# B&R Automation Studio project RobotNewEra (part 10)

### HmiKeyControlGlobal.typ - Program interface
```iecst
(********************************************************************
 * COPYRIGHT -- Bernecker + Rainer
 ********************************************************************
 * Program: HmiKeyControl
 * File: HmiKeyControl.typ
 * Author: B&R, International Applications
 * Created: March 16, 2009
 ********************************************************************
 * Data types of program HmiKeyControl
 ********************************************************************)

TYPE
	HmiKeyControlSpace_typ : 	STRUCT
		Enable : BOOL;
		X1 : REAL;
		Y1 : REAL;
		Z1 : REAL;
		X2 : REAL;
		Y2 : REAL;
		Z2 : REAL;
	END_STRUCT;
	HmiKeyControlInputCommand_Type : 	STRUCT
		StartKey : BOOL; (* Start button has been pressed *)
		StopKey : BOOL; (* Stop button has been pressed *)
		EmergencyStopKey : BOOL;
		PageKey : ARRAY[0..MAX_PAGE_KEY_MINUS_ONE]OF BOOL;
		VirFunctionKeyLeft : ARRAY[0..MAX_FUNCTION_KEY_MINUS_ONE]OF BOOL;
		VirFunctionKey : ARRAY[0..MAX_FUNCTION_KEY_MINUS_ONE]OF BOOL;
		FunctionKey : ARRAY[0..MAX_FUNCTION_KEY_MINUS_ONE]OF BOOL;
		PlusKey : ARRAY[0..MAX_PLUS_MINUS_KEY_MINUS_ONE]OF BOOL;
		MinusKey : ARRAY[0..MAX_PLUS_MINUS_KEY_MINUS_ONE]OF BOOL;
		KeySwitch : ARRAY[0..1]OF BOOL;
		Key2nd : BOOL;
		ProgramActive : BOOL;
		Acknowledge : BOOL;
		Reset : BOOL;
		JogMode : BOOL;
		JogEnable : BOOL;
		FeedrateChange : BOOL;
		StepOn : BOOL;
		SaftyKeyRight : BOOL;
		SaftyKeyLeft : BOOL;
		SetPC : BOOL;
		FileSelect : BOOL;
		PosSwitch : BOOL;
	END_STRUCT;
	HmiKeyControlInputPara_Type : 	STRUCT
		JogMode : USINT;
		SystemAddress : UDINT;
		CncAddress : UDINT;
		AxesAddress : UDINT;
		JogAddress : UDINT;
		RecipeAddress : UDINT;
		ErrorAddress : UDINT;
		JoystickXValue : DINT;
		JoystickYValue : DINT;
		JoystickZValue : DINT;
	END_STRUCT;
	HmiKeyControlInput_Type : 	STRUCT
		Parameter : HmiKeyControlInputPara_Type;
		Command : HmiKeyControlInputCommand_Type;
	END_STRUCT;
	HmiKeyControlOutputMon_Type : 	STRUCT
		JogJointVelocity : REAL;
		ToolIndex : USINT;
		JogToolIndex : USINT;
		FileName : STRING[32];
		ModuleType : UDINT;
		PosSelect : UINT;
		ShowPos : ARRAY[0..5]OF REAL;
		JogMode : USINT;
	END_STRUCT;
	HmiKeyControlOutput_Type : 	STRUCT
		Monitor : HmiKeyControlOutputMon_Type;
		Status : HmiKeyControlOutputStatus_Type;
	END_STRUCT;
	HmiKeyControlOutputStatus_Type : 	STRUCT
		Enable : USINT;
		Run : BOOL;
		Error : BOOL;
		Moving : BOOL;
		JogEnable : BOOL;
		RealContinue : BOOL;
		MoveStatus : USINT;
		AutoStatus : USINT;
		StatusIconIndex : USINT;
		SwitchMode : USINT;
		SWLimitsIgnored : ARRAY[0..5]OF BOOL;
		MoveAxis : ARRAY[0..5]OF SINT;
	END_STRUCT;
	HmiKeyControlComponentsType : 	STRUCT
		LayerButtons : HmiKeyCtrlLayerButtonsType;
		LayerLogin : HmiKeyCtrlLayerLoginType;
	END_STRUCT;
	HmiKeyCtrlLayerLoginType : 	STRUCT
		Layer : HmiLayerType;
	END_STRUCT;
	HmiKeyCtrlLayerButtonsType : 	STRUCT
		Layer : HmiLayerType;
		Tabs : HmiTabsType;
		ButtonVMinus : HmiButtonType;
		ButtonVPlus : HmiButtonType;
		ButtonSwitchOn : HmiButtonType;
		ButtonLogin : HmiButtonType;
		ButtonJogBase : HmiButtonType;
		ButtonJogTool : HmiButtonType;
		ButtonJogJoint : HmiButtonType;
		ButtonJogDirect : HmiButtonType;
		ButtonSingle : HmiButtonType;
		ButtonCont : HmiButtonType;
		SliderV : HmiSliderType;
		NumericV : HmiNumericType;
	END_STRUCT;
	HmiKeyControl_Type : 	STRUCT
		Input : HmiKeyControlInput_Type;
		Output : HmiKeyControlOutput_Type;
		Components : HmiKeyControlComponentsType;
	END_STRUCT;
END_TYPE
```

### HmiKeyControlGlobal.var
```iecst
(********************************************************************
 * COPYRIGHT -- Bernecker + Rainer
 ********************************************************************
 * Program: HmiKeyControl
 * File: HmiKeyControl.var
 * Author: B&R, International Applications
 * Created: March 16, 2009
 ********************************************************************
 * Variables of program HmiKeyControl
 ********************************************************************)
VAR CONSTANT
	AXIS_STATUS_BACKWARD : USINT := 2;
	AXIS_STATUS_FORWARD : USINT := 1;
	AXIS_STATUS_NOACTIVE : USINT := 0;
	AXIS_STATUS_WARNING : USINT := 3;
	HANDWHEEL_STATUS_ACTIVE : USINT := 1;
	HANDWHEEL_STATUS_HALT : USINT := 2;
	HANDWHEEL_STATUS_NOACTIVE : USINT := 0;
	HMIKEYCONTROL_CHANGEMODEAUTO : UINT := 150;
	HMIKEYCONTROL_CHANGEMODEDRYRUN : UINT := 190;
	HMIKEYCONTROL_CHANGEMODEHOME : UINT := 200;
	HMIKEYCONTROL_CHANGEMODEJOG : UINT := 170;
	HMIKEYCONTROL_CHANGEMODEMDI : UINT := 160;
	HMIKEYCONTROL_CHANGEMODESIMUL : UINT := 210;
	HMIKEYCONTROL_CHANGEMODESINGLE : UINT := 180;
	HMIKEYCONTROL_IDLE : UINT := 100;
	HMIKEYCONTROL_INIT : UINT := 0;
	HMIKEYCONTROL_SELECTAXIS : UINT := 120;
	HMIKEYCONTROL_SELECTFUNCTIONM : UINT := 130;
	HMIKEYCONTROL_SELECTSCALE : UINT := 140;
	HMIKEYCONTROL_SELECTSYSTEM : UINT := 110;
	HMIKEYCONTROL_START : UINT := 220;
	HMIKEYCONTROL_STOPAUTO : UINT := 230;
	HMIKEYCONTROL_STOPDRYRUN : UINT := 231;
	HMIKEYCONTROL_STOPHOME : UINT := 232;
	HMIKEYCONTROL_STOPJOG : UINT := 233;
	HMIKEYCONTROL_STOPMDI : UINT := 234;
	HMIKEYCONTROL_STOPSIMUL : UINT := 235;
	HMIKEYCONTROL_STOPSINGLE : UINT := 236;
	MFUNCTION_M10 : USINT := 10;
	MFUNCTION_M11 : USINT := 11;
	MFUNCTION_M12 : USINT := 12;
	MFUNCTION_M13 : USINT := 13;
	MFUNCTION_M14 : USINT := 14;
	MFUNCTION_M15 : USINT := 15;
	MFUNCTION_M16 : USINT := 16;
	MFUNCTION_M17 : USINT := 17;
	MFUNCTION_COOLING : USINT := 1;
	MFUNCTION_DISABLE : USINT := 2;
	MFUNCTION_RUNNING : USINT := 3;
	MFUNCTION_SPINDLE : USINT := 3;
	MFUNCTION_STANDBY : USINT := 0;
	MFUNCTION_STANDBYRUNNING : USINT := 1;
	MFUNCTION_TIMEPRESSED : TIME := T#2s;
	MFUNCTION_WARNING : USINT := 4;
	MODE_AUTOMATIC : USINT := 0;
	MODE_DRYRUN : USINT := 4;
	MODE_HOME : USINT := 5;
	MODE_MDI : USINT := 1;
	MODE_MOTION_AUTO : USINT := 1;
	MODE_MOTION_JOG : USINT := 0;
	MODE_NOMODE : USINT := 254;
	MODE_SIMULATION : USINT := 6;
	MODE_SINGLESTEP : USINT := 3;
	SCALE_STATUS_ACIVE : BOOL := TRUE;
	SCALE_STATUS_NOACTIVE : BOOL := FALSE;
	SCALE_UNITS_INDEX_0 : REAL := 1.0;
	SCALE_UNITS_INDEX_1 : REAL := 0.1;
	SCALE_UNITS_INDEX_2 : REAL := 0.01;
	SYSTEM_STATUS_NOACTIVE : USINT := 0;
	SYSTEM_STATUS_PROGRAMHALT : USINT := 4;
	SYSTEM_STATUS_RUNNING : USINT := 2;
	SYSTEM_STATUS_SELECTED : USINT := 1;
	SYSTEM_STATUS_SELECTRUNNING : USINT := 3;
	SYSTEM_STATUS_WARNING : USINT := 5;
	JOG_MODE_JOINT : USINT := 0;
	JOG_MODE_BASE : USINT := 1;
	JOG_MODE_TOOL : USINT := 2;
	JOG_MODE_DIRECT : USINT := 3;
	WARNING_TIMEACTIVE : TIME := T#3s;
END_VAR
VAR
	HmiKeyControl : HmiKeyControl_Type := (0);
END_VAR
```

### Program Logical/HmiHandling/HmiKeyCtrl/HmiKeyCtrl (IEC) - Handles the Cnc panel key control  functionalities

#### HmiKeyControlActions.st
```iecst
(*Copy all inputs for this program*)
ACTION HmiKeyControlInputs: //Control all the Inputs

	(* Checks if the Simulation key is active and assignes the commands *)
	IF (HmiKeyControl.Output.Monitor.ModuleType = ARSIM_PC)THEN

		FOR i := 0 TO MAX_FUNCTION_KEY_MINUS_ONE DO
			HmiKeyControl.Input.Command.FunctionKey[i]	:= HmiHardKey.Input.MP50_SimKey[22+i];
		END_FOR

		FOR i := 0 TO MAX_PLUS_MINUS_KEY_MINUS_ONE DO
			HmiKeyControl.Input.Command.PlusKey[i]	:= HmiHardKey.Input.MP50_SimKey[16+i];
		END_FOR

		FOR i := 0 TO MAX_PLUS_MINUS_KEY_MINUS_ONE DO
			HmiKeyControl.Input.Command.MinusKey[i]	:= HmiHardKey.Input.MP50_SimKey[8+i];
		END_FOR

		FOR i := 0 TO MAX_PAGE_KEY_MINUS_ONE DO
			HmiKeyControl.Input.Command.PageKey[i]	:= HmiHardKey.Input.MP50_SimKey[i];
		END_FOR
		HmiKeyControl.Input.Command.PageKey[3] := HmiHardKey.Input.MP50_SimKey[3] OR HmiKeyControl.Input.Command.FileSelect;

		HmiKeyControl.Input.Command.StartKey			:= HmiHardKey.Input.MP50_SimKey[7];
		HmiKeyControl.Input.Command.StopKey 			:= HmiHardKey.Input.MP50_SimKey[15];
		HmiKeyControl.Input.Command.EmergencyStopKey 	:= DI1.I3;
		HmiKeyControl.Input.Command.Key2nd 				:= HmiHardKey.Input.MP50_SimKey[14];
		HmiKeyControl.Input.Command.KeySwitch[JOG] 		:= HmiHardKey.Input.MP50_SimKey[35];
		HmiKeyControl.Input.Command.KeySwitch[AUTO] 	:= HmiHardKey.Input.MP50_SimKey[36];

		HmiKeyControl.Input.Command.SaftyKeyLeft	;
		HmiKeyControl.Input.Command.SaftyKeyRight	;

		HmiKeyControl.Input.Command.SaftyKeyLeft		:= TRUE;
		HmiKeyControl.Input.Command.SaftyKeyRight		:= TRUE;

		HmiHardKey.Input.Joystick_XValue	:= 500;
		HmiHardKey.Input.Joystick_YValue	:= 500;
		HmiHardKey.Input.Joystick_ZValue	:= 500;
	ELSE
		FOR i := 0 TO MAX_FUNCTION_KEY_MINUS_ONE DO
			HmiKeyControl.Input.Command.FunctionKey[i]	:= HmiHardKey.Input.MP50_Key[22+i];
		END_FOR

		FOR i := 0 TO MAX_PLUS_MINUS_KEY_MINUS_ONE DO
			HmiKeyControl.Input.Command.PlusKey[i]	:= HmiHardKey.Input.MP50_Key[16+i];
		END_FOR

		FOR i := 0 TO MAX_PLUS_MINUS_KEY_MINUS_ONE DO
			HmiKeyControl.Input.Command.MinusKey[i]	:= HmiHardKey.Input.MP50_Key[8+i];
		END_FOR

		FOR i := 0 TO MAX_PAGE_KEY_MINUS_ONE DO
			HmiKeyControl.Input.Command.PageKey[i]	:= HmiHardKey.Input.MP50_Key[i];
		END_FOR
		HmiKeyControl.Input.Command.PageKey[3] := HmiHardKey.Input.MP50_Key[3] OR HmiKeyControl.Input.Command.FileSelect;

		HmiKeyControl.Input.Command.StartKey			:= HmiHardKey.Input.MP50_Key[7];
		HmiKeyControl.Input.Command.StopKey 			:= HmiHardKey.Input.MP50_Key[15];
		HmiKeyControl.Input.Command.EmergencyStopKey 	:= DI1.I3;
		HmiKeyControl.Input.Command.Key2nd 				:= HmiHardKey.Input.MP50_Key[14];
		HmiKeyControl.Input.Command.KeySwitch[JOG] 		:= HmiHardKey.Input.MP50_Key[35];
		HmiKeyControl.Input.Command.KeySwitch[AUTO] 	:= HmiHardKey.Input.MP50_Key[36];

		HmiKeyControl.Input.Command.SaftyKeyLeft		:= DI1.I1;
		HmiKeyControl.Input.Command.SaftyKeyRight		:= DI1.I2;

		HmiKeyControl.Input.Command.SaftyKeyLeft		:= TRUE;
		HmiKeyControl.Input.Command.SaftyKeyRight		:= TRUE;
	END_IF

	HmiKeyControl.Input.Parameter.JoystickXValue	:= HmiHardKey.Input.Joystick_XValue;
	HmiKeyControl.Input.Parameter.JoystickYValue	:= HmiHardKey.Input.Joystick_YValue;
	HmiKeyControl.Input.Parameter.JoystickZValue	:= HmiHardKey.Input.Joystick_ZValue;

	//LEDs
	HmiHardKey.Output.Motion_Led 		:= pSystem[0].Output.Status.ControllerStatus <> 0;
	HmiHardKey.Output.Run_Led 			:= 1;
	HmiHardKey.Output.Error_Led 		:= HmiKeyControl.Output.Status.Error;
	HmiHardKey.Output.Process_Led 		:= pCnc[0].Output.State.Moving;

END_ACTION

ACTION HmiKeyControlStateHandling: // Main State Machine

	// Emegency Stop
	IF pSystem[0].Output.State.Errorstop THEN
		Internal.HmiKeyControlState := HMIKEYCONSTATESTEP_ERROR;
	END_IF

	// Switch On/Off Control
	IF HmiKeyControl.Components.LayerButtons.ButtonSwitchOn.Value > HmiKeyControl.Components.LayerButtons.ButtonSwitchOn.OldValue THEN
		IF 	pSystem[0].Output.State.Disabled THEN
			pSystem[0].Input.Command.Enable := 1;
			Internal.HmiKeyControlState := HMIKEYCONSTATESTEP_DISABLED;
		ELSIF pCnc[0].Output.State.Standby THEN
			pSystem[0].Input.Command.Enable := 0;
		END_IF
	END_IF

	CASE Internal.HmiKeyControlState OF

		HMIKEYCONSTATESTEP_DISABLED:

			IF HmiKeyControl.Components.LayerButtons.ButtonSwitchOn.Value > HmiKeyControl.Components.LayerButtons.ButtonSwitchOn.OldValue AND NOT pSystem[0].Output.Status.Busy THEN

				IF 	pSystem[0].Output.State.Disabled THEN
					pSystem[0].Input.Command.Enable := 1;
					Internal.HmiKeyControlState := HMIKEYCONSTATESTEP_HOME;
				ELSIF pCnc[0].Output.State.Standby THEN
					pSystem[0].Input.Command.Enable := 0;
				END_IF

			END_IF

			// If Press Start when disabled, show the warning
			IF (HmiKeyControl.Input.Command.StartKey > Internal.OldCommand.StartKey) THEN

				WarnMessage[0] := 1;

			END_IF

		HMIKEYCONSTATESTEP_HOME: (* Homing Axes *)

			// Do the homing, homing position is stored in the Recipe
			IF NOT pSystem[0].Output.Status.Busy AND pSystem[0].Output.Status.ControllerStatus <> 0 THEN

				FOR i := 6 TO MAX_AX_MINUS_TWO DO
					pAxes[i].Input.Parameter.HomePosition := pRecipe.Data.System.HomePosition[i];
				END_FOR

				pSystem[0].Input.Command.Home := 1;

				Internal.HmiKeyControlState := HMIKEYCONSTATESTEP_CHANGEMODE;

			END_IF

		HMIKEYCONSTATESTEP_CHANGEMODE: (* Actual Standby State(After Homing) *)

			IF NOT pSystem[0].Output.Status.Busy AND pSystem[0].Input.Command.Home = 0 THEN

				// Just to avoid the sw limits being ignored
				FOR i := 6 TO MAX_AX_MINUS_TWO DO

					IF HmiKeyControl.Output.Status.SWLimitsIgnored[i - 6] THEN
						pAxes[i].Input.Parameter.WriteParID := ACP10PAR_SGEN_SW_END_IGNORE;
						pAxes[i].Input.Parameter.WriteParIDText := '0';
						pAxes[i].Input.Command.WriteAxisPar := 1;
					END_IF

					HmiKeyControl.Output.Status.SWLimitsIgnored[i - 6] := FALSE;

				END_FOR

				// Make Sure the robot is homed before mode switch to CNC
				IF HmiRetain.HmiKeyControl.MechHomeOK THEN

					IF HmiKeyControl.Output.Status.SwitchMode = LOCK THEN

						pSystem[0].Input.Parameter.Mode := 1;
						Internal.HmiKeyControlState := HMIKEYCONSTATESTEP_ACTIVE_JOG; // JOG MEANS NO CNC, not the Jog Mode for Robot (This mode is for Setting home position)

					ELSE

						pSystem[0].Input.Parameter.Mode := 0;
						Internal.HmiKeyControlState := HMIKEYCONSTATESTEP_ACTIVE_AUTO; // AUTO MEANS CNC, including Jog Mode and Auto Mode

					END_IF

				ELSE

					pSystem[0].Input.Parameter.Mode := 1;
					Internal.HmiKeyControlState := HMIKEYCONSTATESTEP_ACTIVE_JOG;

				END_IF

				pSystem[0].Input.Command.ChangeMode := 1;

			END_IF

		HMIKEYCONSTATESTEP_ACTIVE_JOG:

			IF pSystem[0].Output.Monitor.Mode = 1 THEN (* 1 for No CNC and 0 for CNC *)

				IF HmiKeyControl.Output.Status.SwitchMode <> LOCK THEN

					IF HmiRetain.HmiKeyControl.MechHomeOK THEN

						pSystem[0].Input.Parameter.Mode := 0;
						pSystem[0].Input.Command.ChangeMode := 1;

						StartState := 0;

						Internal.HmiKeyControlState := HMIKEYCONSTATESTEP_ACTIVE_AUTO;

					END_IF

				END_IF

				// The Moving Of Axis in NON-CNC Mode is only allowed in PAGE_SETUPCALIB
				IF HmiGlobal.PageControl.ActPage = PAGE_SETUPCALIB AND pSystem[0].Output.State.Active THEN

					FOR i := 0 TO 5 DO
						(* For MP50-4*)
						IF HmiSetupCtrl.Components.PageCalib.LayerDefault.ButtonAxisToggle[i].Value = 1 THEN // Only when certain Axis is toggled(only one axis will be toggled at one time)
							// Using MCMoveVelocity(Axis Controlling) for Calibration
							IF EDGEPOS((HmiKeyControl.Input.Command.SaftyKeyLeft OR HmiKeyControl.Input.Command.SaftyKeyRight) AND (HmiKeyControl.Input.Command.PlusKey[i] <> 0)
								) THEN
								pAxes[i+6].Input.Parameter.Velocity := HmiKeyControl.Components.LayerButtons.SliderV.Value /100.0 * pRecipe.Data.System.JointJogSpeed;
								pAxes[i+6].Input.Parameter.Direction := mcPOSITIVE_DIR;
								pAxes[i+6].Input.Command.MoveVelocity := 1;
							ELSIF EDGENEG((HmiKeyControl.Input.Command.SaftyKeyLeft OR HmiKeyControl.Input.Command.SaftyKeyRight) AND (HmiKeyControl.Input.Command.PlusKey[i] <> 0)
								) THEN
								pAxes[i+6].Input.Command.Stop := 1;
							ELSIF EDGEPOS((HmiKeyControl.Input.Command.SaftyKeyLeft OR HmiKeyControl.Input.Command.SaftyKeyRight) AND (HmiKeyControl.Input.Command.MinusKey[i] <> 0)
								) THEN
								pAxes[i+6].Input.Parameter.Velocity := HmiKeyControl.Components.LayerButtons.SliderV.Value /100.0 * pRecipe.Data.System.JointJogSpeed;
								pAxes[i+6].Input.Parameter.Direction := mcNEGATIVE_DIR;
								pAxes[i+6].Input.Command.MoveVelocity := 1;
							ELSIF EDGENEG((HmiKeyControl.Input.Command.SaftyKeyLeft OR HmiKeyControl.Input.Command.SaftyKeyRight) AND (HmiKeyControl.Input.Command.MinusKey[i] <> 0)
								) THEN
								pAxes[i+6].Input.Command.Stop := 1;

							END_IF
						ELSE

							// Otherweise stop the Movement
							IF pAxes[i+6].Output.State.ContinuousMotion THEN

								pAxes[i+6].Input.Command.Stop := 1;

							END_IF
						END_IF

					END_FOR

				ELSE
					// In other Page stop the Axis Any Way
					FOR i := 0 TO 5 DO
						IF pAxes[i+6].Output.State.ContinuousMotion THEN

							pAxes[i+6].Input.Command.Stop := 1;

						END_IF
					END_FOR
				END_IF

			END_IF

		HMIKEYCONSTATESTEP_ACTIVE_AUTO:  // CNC Mode

			IF pSystem[0].Output.Monitor.Mode = 0 THEN
				// Change to Non-CNC Mode
				IF HmiKeyControl.Output.Status.SwitchMode = LOCK THEN

					pSystem[0].Input.Parameter.Mode := 1;
					pSystem[0].Input.Command.ChangeMode := 1;

					Internal.HmiKeyControlState := HMIKEYCONSTATESTEP_ACTIVE_JOG;

				END_IF

				(* UserLevel higher than 0 and Mode is Auto then Start OR Stop is allowed *)
				IF pSystem[0].Output.State.Active AND gUserLevel > 0 AND HmiKeyControl.Output.Status.MoveStatus = AUTO THEN

					pCnc[0].Input.Parameter.NcInitProgramName := '';

					(* Stop the Program: Once for Halt, Twice for Stop *)
					IF HmiKeyControl.Input.Command.StopKey > Internal.OldCommand.StopKey THEN

						IF pCnc[0].Output.State.Moving AND NOT pCnc[0].Output.Status.Halted THEN
							pCnc[0].Input.Command.Halt := 1;
						ELSE
							pCnc[0].Input.Command.Stop := 1;
						END_IF

					END_IF

					// Start the program
					IF (HmiKeyControl.Input.Command.StartKey > Internal.OldCommand.StartKey) THEN

						(* if halted continue else start *)
						IF pCnc[0].Output.Status.Halted THEN
							pCnc[0].Input.Command.Continue := 1;
						ELSE

							IF HmiRetain.HmiProgram.Name <> ''  THEN
								IF HmiRetain.HmiProgram.Ptr <> 0 THEN // Start the Program from some line (Not working right now)
									brsitoa(HmiRetain.HmiProgram.Ptr, ADR(TempStr));
									pCnc[0].Input.Parameter.NcProgramName := CONCAT(CONCAT(CONCAT(HmiRetain.HmiProgram.Name, '.st'), '::'), TempStr);
								ELSE
									pCnc[0].Input.Parameter.NcProgramName := CONCAT(HmiRetain.HmiProgram.Name, '.st');
								END_IF

								pCnc[0].Input.Parameter.NcProgramStartPos := -1;
								pCnc[0].Input.Parameter.NcProgramStartMode := ncFILE;
								pCnc[0].Input.Command.StartNcProgram := 1;

							END_IF
						END_IF

					END_IF

					//If Program is stopped, reset the Pointer
					IF EDGENEG(pCnc[0].Output.State.Moving) THEN

						HmiRetain.HmiProgram.Ptr := 0;

					END_IF

				END_IF

			ELSIF pSystem[0].Output.State.Standby AND pSystem[0].Output.Status.HomingOk THEN

				Internal.HmiKeyControlState := HMIKEYCONSTATESTEP_CHANGEMODE;

			END_IF

		HMIKEYCONSTATESTEP_ERROR:
			// Press the Stop key in Error state means reset the error
			IF (HmiKeyControl.Input.Command.StopKey > Internal.OldCommand.StopKey) THEN
				pSystem[0].Input.Command.Reset := 1;
			END_IF

			pCncDat ACCESS pCnc[0].Output.Monitor.CncAddress;

			(* In Case Cnc Still Runing even in Errorstop State *)
			IF (pCncDat.move.status.cnt_ncprog <> 0) THEN
				ncaction(ADR(pCncDat), ncMOVE, ncSTOP);
			END_IF

			IF NOT pSystem[0].Output.State.Errorstop THEN
				IF pSystem[0].Output.Status.HomingOk THEN
					Internal.HmiKeyControlState := HMIKEYCONSTATESTEP_CHANGEMODE;
				ELSE
					Internal.HmiKeyControlState := HMIKEYCONSTATESTEP_HOME;
				END_IF

			END_IF

	END_CASE

	// SingleStep Control
	IF pCnc[0].Output.State.Standby THEN
		(* Switch between Modes: *)
		IF (HmiKeyControl.Components.LayerButtons.ButtonSingle.Value > HmiKeyControl.Components.LayerButtons.ButtonSingle.OldValue) THEN
			IF NOT pCnc[0].Output.Status.SingleStep THEN
				pCnc[0].Input.Command.StartSingleStep := 1;
			END_IF
		END_IF

		IF (HmiKeyControl.Components.LayerButtons.ButtonCont.Value > HmiKeyControl.Components.LayerButtons.ButtonCont.OldValue) THEN
			IF pCnc[0].Output.Status.SingleStep THEN
				pCnc[0].Input.Command.StopSingleStep := 1;
			END_IF
		END_IF

		// Switch off Single Step for Jog
		IF HmiKeyControl.Output.Status.MoveStatus = JOG AND pCnc[0].Output.Status.SingleStep THEN
			pCnc[0].Input.Command.StopSingleStep := 1;
		END_IF

	END_IF
	// Show different Pics
	HmiKeyControl.Components.LayerButtons.Tabs.ButtonsTab[0].BmpIdx := pCnc[0].Output.Status.SingleStep;

END_ACTION

ACTION HmiKeyControlJog: // Jog Control

	IF gUserLevel = 0 THEN

		pJog.Run 	:= 0;

	ELSE
		// Four Modes Available: TOOL; BASE; JOINT; DIRECT
		IF pCnc[0].Output.State.Standby THEN
			(* Switch between Modes *)
			IF HmiKeyControl.Components.LayerButtons.ButtonJogTool.Value > HmiKeyControl.Components.LayerButtons.ButtonJogTool.OldValue THEN
				HmiKeyControl.Input.Parameter.JogMode := JOG_MODE_TOOL;
			END_IF

			IF HmiKeyControl.Components.LayerButtons.ButtonJogBase.Value > HmiKeyControl.Components.LayerButtons.ButtonJogBase.OldValue THEN
				HmiKeyControl.Input.Parameter.JogMode := JOG_MODE_BASE;
			END_IF

			IF HmiKeyControl.Components.LayerButtons.ButtonJogJoint.Value > HmiKeyControl.Components.LayerButtons.ButtonJogJoint.OldValue THEN
				HmiKeyControl.Input.Parameter.JogMode := JOG_MODE_JOINT;
			END_IF

			IF HmiKeyControl.Components.LayerButtons.ButtonJogDirect.Value > HmiKeyControl.Components.LayerButtons.ButtonJogDirect.OldValue THEN
				HmiKeyControl.Input.Parameter.JogMode := JOG_MODE_DIRECT;
			END_IF

		END_IF
		// Show Different Pics
		HmiKeyControl.Components.LayerButtons.Tabs.ButtonsTab[2].BmpIdx := HmiKeyControl.Input.Parameter.JogMode;

		// Buttons Control (+/- Buttons) Plus/Minuskey -> MoveAxis
		IF HmiKeyControl.Output.Status.MoveStatus = JOG THEN

			FOR i := 0 TO 5 DO
				(* For MP50-4*)
				IF (HmiKeyControl.Input.Command.PlusKey[i] <> 0)  THEN
					HmiKeyControl.Output.Status.MoveAxis[i] := 1;
				ELSIF (HmiKeyControl.Input.Command.MinusKey[i] <> 0) THEN
					HmiKeyControl.Output.Status.MoveAxis[i] := -1;
				ELSE
					HmiKeyControl.Output.Status.MoveAxis[i] := 0;
				END_IF

			END_FOR

			IF (HmiKeyControl.Input.Command.SaftyKeyLeft = 0)
				AND (HmiKeyControl.Input.Command.SaftyKeyRight = 0) THEN

				HmiKeyControl.Output.Status.MoveAxis[0] := 0;
				HmiKeyControl.Output.Status.MoveAxis[1] := 0;
				HmiKeyControl.Output.Status.MoveAxis[2] := 0;
				HmiKeyControl.Output.Status.MoveAxis[3] := 0;
				HmiKeyControl.Output.Status.MoveAxis[4] := 0;
				HmiKeyControl.Output.Status.MoveAxis[5] := 0;
			END_IF

			IF (HmiKeyControl.Output.Status.MoveAxis[0] <> 0) OR
				(HmiKeyControl.Output.Status.MoveAxis[1] <> 0) OR
				(HmiKeyControl.Output.Status.MoveAxis[2] <> 0) OR
				(HmiKeyControl.Output.Status.MoveAxis[3] <> 0) OR
				(HmiKeyControl.Output.Status.MoveAxis[4] <> 0) OR
				(HmiKeyControl.Output.Status.MoveAxis[5] <> 0) THEN

				IF (pRecipe.Data.System.JointJogSpeed <> 0) THEN

					IF (HmiKeyControl.Input.Parameter.JogMode = JOG_MODE_BASE) THEN
						pJog.Speed 	:= pRecipe.Data.System.PathJogSpeed;

					ELSIF (HmiKeyControl.Input.Parameter.JogMode = JOG_MODE_TOOL) THEN
						pJog.Speed 	:= pRecipe.Data.System.PathJogSpeed;

					ELSIF (HmiKeyControl.Input.Parameter.JogMode = JOG_MODE_JOINT) THEN
						pJog.Speed 	:= pRecipe.Data.System.JointJogSpeed;
					END_IF

					pJog.Mode	:= HmiKeyControl.Input.Parameter.JogMode;
					pJog.Run 	:= 1;

				END_IF

			ELSE

				// Special Control For Direct Mode
				IF (HmiKeyControl.Input.Command.SaftyKeyLeft = 1 OR HmiKeyControl.Input.Command.SaftyKeyRight = 1) AND
					HmiKeyControl.Input.Parameter.JogMode = JOG_MODE_DIRECT AND HmiGlobal.PageControl.ActPage = PAGE_JOGGING AND
					HmiJog.Components.LayerDefault.TextActSet.TextIndex = 1 THEN // The use of this mode is restricted to certain page and certain status

					IF HmiJog.Components.LayerDefault.ButtonCheckVar.Value = 0 THEN // Use the point from numeric inputs.
						IF HmiJog.Components.LayerDefault.DropdownJointTCP.SelectedIndex = 0 THEN

							pJog.Speed := pRecipe.Data.System.JointJogSpeed;

							JointSync.JointAxis[0] := HmiJog.Components.LayerDefault.NumericPosSet[0].Value;
							JointSync.JointAxis[1] := HmiJog.Components.LayerDefault.NumericPosSet[1].Value;
							JointSync.JointAxis[2] := HmiJog.Components.LayerDefault.NumericPosSet[2].Value;
							JointSync.JointAxis[3] := HmiJog.Components.LayerDefault.NumericPosSet[3].Value;
							JointSync.JointAxis[4] := HmiJog.Components.LayerDefault.NumericPosSet[4].Value;
							JointSync.JointAxis[5] := HmiJog.Components.LayerDefault.NumericPosSet[5].Value;

							JointTCPSync := 1;

						ELSE
							pJog.Speed := pRecipe.Data.System.PathJogSpeed;

							PointSync.Pos.x := HmiJog.Components.LayerDefault.NumericPosSet[0].Value;
							PointSync.Pos.y := HmiJog.Components.LayerDefault.NumericPosSet[1].Value;
							PointSync.Pos.z := HmiJog.Components.LayerDefault.NumericPosSet[2].Value;
							PointSync.Orient.Angle[0] := HmiJog.Components.LayerDefault.NumericPosSet[3].Value;
							PointSync.Orient.Angle[1] := HmiJog.Components.LayerDefault.NumericPosSet[4].Value;
							PointSync.Orient.Angle[2] := HmiJog.Components.LayerDefault.NumericPosSet[5].Value;
							PointSync.Orient.Angle[3] := HmiJog.Components.LayerDefault.NumericPosSet[6].Value;

							IF HmiJog.Components.LayerDefault.DropdownEulerQuan.SelectedIndex = 1 THEN
								PointSync.Orient.Type := MX_QUATERNION;
							ELSE
								PointSync.Orient.Type := 1;
							END_IF

							JointTCPSync := 0;
						END_IF
					ELSE
						// Else use the Point from the File
						IF HmiRetain.HmiJog.Device = HmiRetain.HmiEditor.Device AND HmiRetain.HmiJog.Name = HmiRetain.HmiEditor.Name THEN

							IF HmiRetain.HmiJog.Joint.Set THEN

								pJog.Speed := pRecipe.Data.System.JointJogSpeed;

								JointSync := HmiRetain.HmiJog.Joint.Joint;

								JointTCPSync := 1;

							END_IF

							IF HmiRetain.HmiJog.Point.Set THEN

								pJog.Speed := pRecipe.Data.System.PathJogSpeed;

								PointSync := HmiRetain.HmiJog.Point.Point;

								JointTCPSync := 0;

							END_IF

						END_IF

					END_IF

					pJog.Mode	:= HmiKeyControl.Input.Parameter.JogMode;

					pJog.Run 	:= 1;

				ELSE

					pJog.Run	:= 0;

				END_IF

			END_IF

		END_IF

	END_IF

END_ACTION

ACTION HmiKeyControlStatus:

	// Control all the status, altogether 4  stats(Disabled/LOCK/JOG/AUTO)
	IF HmiKeyControl.Input.Command.KeySwitch[JOG] THEN
		HmiKeyControl.Output.Status.SwitchMode := JOG;
	ELSIF HmiKeyControl.Input.Command.KeySwitch[AUTO] THEN
		HmiKeyControl.Output.Status.SwitchMode := AUTO;
	ELSE
		HmiKeyControl.Output.Status.SwitchMode := LOCK;
	END_IF

	IF pSystem[0].Output.State.Disabled THEN // Not Enabled = DISABLED
		HmiKeyControl.Output.Status.MoveStatus := DISABLED;
	ELSE
		IF pSystem[0].Output.Monitor.Mode = 1 THEN // If in the middle, Lock
			HmiKeyControl.Output.Status.MoveStatus := LOCK;
		ELSIF pSystem[0].Output.Monitor.Mode = 0 THEN // Left Jog
			IF HmiKeyControl.Output.Status.SwitchMode = AUTO THEN
				HmiKeyControl.Output.Status.MoveStatus := AUTO;
			ELSE // Right Auto
				HmiKeyControl.Output.Status.MoveStatus := JOG;
			END_IF

		END_IF

	END_IF
	// In AutoMode 3 Status(RUN/PAUSE/STOP)
	IF (HmiKeyControl.Output.Status.MoveStatus = AUTO) THEN
		IF (pCnc[0].Output.State.Moving = 1) AND (pCnc[0].Output.Status.Halted  = 0) THEN
			HmiKeyControl.Output.Status.AutoStatus := RUN;
		ELSIF (pCnc[0].Output.State.Moving = 1) AND (pCnc[0].Output.Status.Halted  = 1) THEN
			HmiKeyControl.Output.Status.AutoStatus := PAUSE;
		ELSE
			HmiKeyControl.Output.Status.AutoStatus := STOP;
		END_IF
	ELSE
		HmiKeyControl.Output.Status.AutoStatus := STOP;
	END_IF

END_ACTION

ACTION HmiKeyControlPage:
	// Turn the Pages
	IF (HmiKeyControl.Input.Command.PageKey[0] > Internal.OldCommand.PageKey[0]) THEN
		HmiGlobal.PageControl.SetPage := PAGE_MAIN;
	END_IF

	IF (HmiKeyControl.Input.Command.PageKey[1] > Internal.OldCommand.PageKey[1]) AND (gUserLevel >= 1) THEN
		HmiGlobal.PageControl.SetPage := PAGE_SETUP;
	END_IF

	IF (HmiKeyControl.Input.Command.PageKey[2] > Internal.OldCommand.PageKey[2]) AND (gUserLevel >= 1) THEN
		HmiGlobal.PageControl.SetPage := PAGE_IO;
	END_IF

	IF (HmiKeyControl.Input.Command.PageKey[3] > Internal.OldCommand.PageKey[3]) AND (gUserLevel >= 1) THEN
		HmiGlobal.PageControl.SetPage := PAGE_PROGRAM;
	END_IF

	// Edit Page cannot be entered if no Program available
	IF (HmiKeyControl.Input.Command.PageKey[4] > Internal.OldCommand.PageKey[4]) AND (gUserLevel >= 1) AND
		HmiRetain.HmiEditor.Device <> '' AND HmiRetain.HmiEditor.Name <> ''  THEN
		HmiGlobal.PageControl.SetPage := PAGE_EDITOR;
	END_IF

	IF (HmiKeyControl.Input.Command.PageKey[5] > Internal.OldCommand.PageKey[5]) AND (gUserLevel >= 1) THEN
		HmiGlobal.PageControl.SetPage := PAGE_JOGGING;
	END_IF

	IF (HmiKeyControl.Input.Command.PageKey[6] > Internal.OldCommand.PageKey[6]) AND (gUserLevel >= 1) THEN
		HmiGlobal.PageControl.SetPage := PAGE_ALARM;
	END_IF

	// If userlevel < 1, robot is disabled
	IF (gUserLevel < 1) THEN

		HmiKeyControl.Components.LayerButtons.ButtonSwitchOn.Value := 0;

	END_IF

	IF HmiKeyControl.Components.LayerButtons.ButtonLogin.Value > HmiKeyControl.Components.LayerButtons.ButtonLogin.OldValue THEN

		HmiKeyControl.Components.LayerLogin.Layer.StatusDatapoint := 0;

	END_IF

END_ACTION

ACTION HmiKeyControlFeedOverride:

	// Using 1st Order Filter to smoothe the Feedrate to avoid rash change.
	LCRPT1_0(enable := 1 , x := HmiKeyControl.Components.LayerButtons.SliderV.Value / 100.0, t := 1); // Time constant 1 second
	pCnc[0].Input.Parameter.FeedrateOverride := LCRPT1_0.y;
	pCnc[0].Input.Parameter.RapidOverride		:= pCnc[0].Input.Parameter.FeedrateOverride;

	// Visual Effect of Slider of Feedrate
	IF NOT pCnc[0].Output.State.Moving OR pCnc[0].Output.Status.Halted THEN
		HmiKeyControl.Components.LayerButtons.SliderV.StatusDatapoint := BIT_SET(HmiKeyControl.Components.LayerButtons.SliderV.StatusDatapoint, 1);
	ELSE
		HmiKeyControl.Components.LayerButtons.SliderV.StatusDatapoint := BIT_CLR(HmiKeyControl.Components.LayerButtons.SliderV.StatusDatapoint, 1);
	END_IF

	(* Delicate control of Plus/Minus Button --- Done by Others(MB Kai YH) *)
	IF (HmiKeyControl.Components.LayerButtons.ButtonVPlus.Value > HmiKeyControl.Components.LayerButtons.ButtonVPlus.OldValue) THEN
		HmiKeyControl.Components.LayerButtons.SliderV.Value := HmiKeyControl.Components.LayerButtons.SliderV.Value + 1;
		VPlus1T := VPlus1T + cycT;
		VPlus10T := VPlus10T + cycT;
	ELSIF (HmiKeyControl.Components.LayerButtons.ButtonVPlus.Value <> 0)
		AND (HmiKeyControl.Components.LayerButtons.ButtonVPlus.OldValue <> 0) THEN
		VPlus1T := VPlus1T + cycT;
		VPlus10T := VPlus10T + cycT;

		IF (VPlus10T > (10*CalculateInterval))
			AND (VPlus1T > CalculateInterval / 3) THEN
			HmiKeyControl.Components.LayerButtons.SliderV.Value := HmiKeyControl.Components.LayerButtons.SliderV.Value + 1;
			VPlus1T := 0;
		ELSIF (VPlus1T > CalculateInterval)THEN
			HmiKeyControl.Components.LayerButtons.SliderV.Value := HmiKeyControl.Components.LayerButtons.SliderV.Value + 1;
			VPlus1T := 0;
		END_IF
	ELSIF (HmiKeyControl.Components.LayerButtons.ButtonVMinus.Value > HmiKeyControl.Components.LayerButtons.ButtonVMinus.OldValue) THEN
		HmiKeyControl.Components.LayerButtons.SliderV.Value := HmiKeyControl.Components.LayerButtons.SliderV.Value - 1;
		VPlus1T := VPlus1T + cycT;
		VPlus10T := VPlus10T + cycT;
	ELSIF (HmiKeyControl.Components.LayerButtons.ButtonVMinus.Value <> 0)
		AND (HmiKeyControl.Components.LayerButtons.ButtonVMinus.OldValue <> 0) THEN
		VPlus1T := VPlus1T + cycT;
		VPlus10T := VPlus10T + cycT;
		IF (VPlus10T > (10*CalculateInterval))
			AND (VPlus1T > CalculateInterval / 3) THEN
			HmiKeyControl.Components.LayerButtons.SliderV.Value := HmiKeyControl.Components.LayerButtons.SliderV.Value - 1;
			VPlus1T := 0;
		ELSIF (VPlus1T > CalculateInterval)THEN
			HmiKeyControl.Components.LayerButtons.SliderV.Value := HmiKeyControl.Components.LayerButtons.SliderV.Value - 1;
			VPlus1T := 0;
		END_IF
	ELSE
		CalculateInterval := 500;
		VPlus1T := 0;
		VPlus10T:= 0;
	END_IF

	// Set the Limit of SliderV (Feedrate)
	IF (HmiKeyControl.Components.LayerButtons.SliderV.Value > 100) THEN
		HmiKeyControl.Components.LayerButtons.SliderV.Value := 100;
	ELSIF (HmiKeyControl.Components.LayerButtons.SliderV.Value < 1) THEN
		HmiKeyControl.Components.LayerButtons.SliderV.Value := 1;
	END_IF

END_ACTION

ACTION HmiKeyControlVisuHandling:

	// Visu Handling for Common Layer including Tabs (Cont/Singlestep Feedrate JogMode etc)
	FOR i := 0 TO HmiKeyControl.Components.LayerButtons.Tabs.TabMaxIndex DO
		IF HmiKeyControl.Components.LayerButtons.Tabs.ButtonsTab[i].Value > HmiKeyControl.Components.LayerButtons.Tabs.ButtonsTab[i].OldValue THEN
			FOR j := 0 TO HmiKeyControl.Components.LayerButtons.Tabs.TabMaxIndex DO
				IF j <> i THEN
					HmiKeyControl.Components.LayerButtons.Tabs.ButtonsTab[j].Value := 0;
				END_IF
			END_FOR
		END_IF
	END_FOR

	HmiKeyControl.Components.LayerButtons.Tabs.TabBg.StatusDatapoint := 1;

	FOR i := 0 TO HmiKeyControl.Components.LayerButtons.Tabs.TabMaxIndex DO
		IF HmiKeyControl.Components.LayerButtons.Tabs.ButtonsTab[i].Value = 1 THEN
			HmiKeyControl.Components.LayerButtons.Tabs.ButtonsTab[i].StatusDatapoint := BIT_CLR(HmiKeyControl.Components.LayerButtons.Tabs.ButtonsTab[i].StatusDatapoint, 0);
			HmiKeyControl.Components.LayerButtons.Tabs.TabSelectedIndex := i;
			HmiKeyControl.Components.LayerButtons.Tabs.TabBg.StatusDatapoint := 0;
		ELSE
			HmiKeyControl.Components.LayerButtons.Tabs.ButtonsTab[i].StatusDatapoint := BIT_SET(HmiKeyControl.Components.LayerButtons.Tabs.ButtonsTab[i].StatusDatapoint, 0);
		END_IF
	END_FOR

	IF HmiKeyControl.Output.Status.MoveStatus = AUTO THEN
		HmiKeyControl.Components.LayerButtons.Tabs.ButtonsTab[0].StatusDatapoint := BIT_CLR(HmiKeyControl.Components.LayerButtons.Tabs.ButtonsTab[0].StatusDatapoint, 1);
	ELSE
		HmiKeyControl.Components.LayerButtons.Tabs.ButtonsTab[0].StatusDatapoint := BIT_SET(HmiKeyControl.Components.LayerButtons.Tabs.ButtonsTab[0].StatusDatapoint, 1);
	END_IF

	IF HmiKeyControl.Output.Status.MoveStatus = JOG THEN
		HmiKeyControl.Components.LayerButtons.Tabs.ButtonsTab[2].StatusDatapoint := BIT_CLR(HmiKeyControl.Components.LayerButtons.Tabs.ButtonsTab[2].StatusDatapoint, 1);
	ELSE
		HmiKeyControl.Components.LayerButtons.Tabs.ButtonsTab[2].StatusDatapoint := BIT_SET(HmiKeyControl.Components.LayerButtons.Tabs.ButtonsTab[2].StatusDatapoint, 1);
	END_IF

	// Login Popu automatically
	IF gUserLevel < 1 THEN
		HmiKeyControl.Components.LayerLogin.Layer.StatusDatapoint := 0;
	END_IF

	// Buttons PosEdge Detection
	HmiKeyControl.Components.LayerButtons.ButtonCont.OldValue := HmiKeyControl.Components.LayerButtons.ButtonCont.Value;
	HmiKeyControl.Components.LayerButtons.ButtonSingle.OldValue := HmiKeyControl.Components.LayerButtons.ButtonSingle.Value;
	HmiKeyControl.Components.LayerButtons.ButtonJogBase.OldValue := HmiKeyControl.Components.LayerButtons.ButtonJogBase.Value;
	HmiKeyControl.Components.LayerButtons.ButtonJogTool.OldValue := HmiKeyControl.Components.LayerButtons.ButtonJogTool.Value;
	HmiKeyControl.Components.LayerButtons.ButtonJogJoint.OldValue := HmiKeyControl.Components.LayerButtons.ButtonJogJoint.Value;
	HmiKeyControl.Components.LayerButtons.ButtonJogDirect.OldValue := HmiKeyControl.Components.LayerButtons.ButtonJogDirect.Value;

	FOR i:= 0 TO HmiKeyControl.Components.LayerButtons.Tabs.TabMaxIndex DO
		HmiKeyControl.Components.LayerButtons.Tabs.ButtonsTab[i].OldValue := HmiKeyControl.Components.LayerButtons.Tabs.ButtonsTab[i].Value;
	END_FOR

	HmiKeyControl.Components.LayerButtons.ButtonLogin.OldValue :=  HmiKeyControl.Components.LayerButtons.ButtonLogin.Value;
	HmiKeyControl.Components.LayerButtons.ButtonSwitchOn.OldValue :=  HmiKeyControl.Components.LayerButtons.ButtonSwitchOn.Value;
	HmiKeyControl.Components.LayerButtons.ButtonVPlus.OldValue :=  HmiKeyControl.Components.LayerButtons.ButtonVPlus.Value;
	HmiKeyControl.Components.LayerButtons.ButtonVMinus.OldValue :=  HmiKeyControl.Components.LayerButtons.ButtonVMinus.Value;

END_ACTION
```

#### HmiKeyControlCyclic.st - Program implementation
```iecst
(************************************************************************************************************************)
(* COPYRIGHT -- Bernecker + Rainer																						*)
(************************************************************************************************************************)
(* Object name: 		HmiKeyControlCyclic																				*)
(* Author:      		B&R																								*)
(* Site:        		Eggelsberg , International Applications                                                       	*)
(* Created:     		February 25, 2009                                                                              	*)
(* Restriction: 		consider task order;								      		                              	*)
(* Description: 		Implementation of the HmiKeyControl													            *)
(*----------------------------------------------------------------------------------------------------------------------*)
(* Version History:		1.00	February 25, 2009																  		*)
(*----------------------------------------------------------------------------------------------------------------------*)
(* Development tool: 	B&R Automation Studio V3.0.80.19 															  	*)
(*----------------------------------------------------------------------------------------------------------------------*)
(* Dependencies: 											                               						       	*)
(************************************************************************************************************************)
PROGRAM _CYCLIC

	hmiRTInfo(enable := 1);
	cycT := hmiRTInfo.cycle_time / 1000;

	IF	(HmiGlobal.Address.AxesAddress <> 0)
		AND	(HmiGlobal.Address.CncAddress <> 0)
		AND	(HmiGlobal.Address.SystemAddress <> 0)
		AND (HmiGlobal.Address.JogAddress <> 0)
		AND	(HmiGlobal.Address.RecipeAddress <> 0)
		AND	(HmiGlobal.Address.ErrorAddress <> 0) THEN

		pAxes ACCESS HmiGlobal.Address.AxesAddress;
		pCnc ACCESS HmiGlobal.Address.CncAddress;
		pSystem ACCESS HmiGlobal.Address.SystemAddress;
		pJog ACCESS HmiGlobal.Address.JogAddress;
		pRecipe ACCESS HmiGlobal.Address.RecipeAddress;
		pError ACCESS HmiGlobal.Address.ErrorAddress;

	ELSE
		RETURN;
	END_IF

	NumberOfActiveSys := 0;

	FOR i:=0 TO MAX_SYS_MINUS_ONE DO
		IF pSystem[i].Input.Configuration.Active THEN
			NumberOfActiveSys  := NumberOfActiveSys + 1;
		END_IF
	END_FOR;

	IF NumberOfActiveSys < MAX_SYS THEN
		RETURN;
	END_IF

	HmiKeyControlInputs;
	HmiKeyControlPage;
	HmiKeyControlStatus;
	HmiKeyControlStateHandling;
	HmiKeyControlJog;
	HmiKeyControlFeedOverride;
	HmiKeyControlVisuHandling;

	Internal.OldCommand := HmiKeyControl.Input.Command;

END_PROGRAM

PROGRAM _EXIT

	brsmemset(ADR(HmiKeyControl),0,SIZEOF(HmiKeyControl));

END_PROGRAM
```

#### HmiKeyControlInit.st - Program implementation
```iecst
(************************************************************************************************************************)
(* COPYRIGHT -- Bernecker + Rainer																						*)
(************************************************************************************************************************)
(* Object name: 		HmiKeyControlCyclic																				*)
(* Author:      		B&R																								*)
(* Site:        		Eggelsberg , International Applications                                                       	*)
(* Created:     		February 25, 2009                                                                              	*)
(* Restriction: 		consider task order;								      		                              	*)
(* Description: 		Implementation of the HmiKeyControl													            *)
(*----------------------------------------------------------------------------------------------------------------------*)
(* Version History:		1.00	February 25, 2009																  		*)
(*----------------------------------------------------------------------------------------------------------------------*)
(* Development tool: 	B&R Automation Studio V3.0.80.19 															  	*)
(*----------------------------------------------------------------------------------------------------------------------*)
(* Dependencies: 											                               						       	*)
(************************************************************************************************************************)
PROGRAM _INIT

	TrfDataAdd := ADR(Robot_TRF);

	HmiKeyControl.Components.LayerLogin.Layer.StatusDatapoint := 0;
	HmiKeyControl.Components.LayerButtons.SliderV.Value := 5;
	FOR i:= 0 TO 4 DO
		HmiKeyControl.Components.LayerButtons.Tabs.ButtonsTab[i].StatusDatapoint := 1;
	END_FOR
	HmiKeyControl.Components.LayerButtons.Tabs.TabMaxIndex := 2;

	HmiKeyControl.Output.Monitor.PosSelect := 0;

	HWInfo_01.enable := 1;     (* Function block only executed if ENABLE <> 0 *)
	HWInfo_01.first := 1;     (* Determines the hardware module that the FUNCTION should be applied TO *)
	HWInfo_01.pName := ADR(HWInfo_01_String);
	HWInfo_01();
	HmiKeyControl.Output.Monitor.ModuleType	:= HWInfo_01.module_typ;
	(* To Delete *)
	//	HmiKeyControl.Output.Monitor.ModuleType := ARSIM_PC;

END_PROGRAM
```

#### HmiKeyControlPrv.var - Local variables
```iecst
(********************************************************************
 * COPYRIGHT -- Bernecker + Rainer
 ********************************************************************
 * Program: HmiKeyControl
 * File: HmiKeyControl.var
 * Author: B&R, International Applications
 * Created: March 16, 2009
 ********************************************************************
 * Local variables of program HmiKeyControl
 ********************************************************************)
VAR CONSTANT
END_VAR
(*Variables*)
VAR
	Internal : HmiKeyCtrlInternal_Type := (0);
END_VAR
(*References*)
VAR
	pAxes : REFERENCE TO ARRAY[0..MAX_AX_MINUS_ONE] OF Axes_Type;
	pCnc : REFERENCE TO ARRAY[0..MAX_CNC_MINUS_ONE] OF Cnc_Type;
	pSystem : REFERENCE TO ARRAY[0..MAX_SYS_MINUS_ONE] OF System_Type;
	pJog : REFERENCE TO Jog_Type;
	pRecipe : REFERENCE TO RECIPE_typ;
	pError : REFERENCE TO Error_Type;
	pCncDat : REFERENCE TO ARNC0CNC_typ;
END_VAR
(*Separator*)
VAR
	j : USINT := 0;
	i : USINT;
	NumberOfActiveSys : USINT;
	hmiRTInfo : RTInfo;
	cycT : DINT;
	CalculateInterval : DINT;
	VPlus1T : DINT;
	VPlus10T : DINT;
	HWInfo_01 : HWInfo;
	HWInfo_01_String : STRING[20];
	TrfDataAdd : UDINT := 0;
	SimPos : ARRAY[0..5] OF REAL;
	StartState : INT;
	TempStr : STRING[5] := '';
	LCRPT1_0 : LCRPT1;
END_VAR
```

#### HmiKeyControlPrv.typ - Program interface
```iecst
(********************************************************************
 * COPYRIGHT -- Bernecker + Rainer
 ********************************************************************
 * Program: HmiKeyControl
 * File: HmiKeyControl.typ
 * Author: B&R, International Applications
 * Created: March 16, 2009
 ********************************************************************
 * Data types of program HmiKeyControl
 ********************************************************************)

TYPE
	MatrixOut_typ : 	STRUCT
		phi : LREAL;
		theta : LREAL;
		psi : LREAL;
	END_STRUCT;
	MatrixRow_typ : 	STRUCT
		Line : ARRAY[0..2]OF LREAL;
	END_STRUCT;
	RotationMatrixInput_typ : 	STRUCT
		M1 : ARRAY[0..2]OF MatrixRow_typ;
		measure : UDINT;
		angles_type : UDINT;
		epsilon : LREAL;
		desired_phi : LREAL;
		desired_theta : LREAL;
		desired_psi : LREAL;
	END_STRUCT;
	HmiKeyControlStateSteps_Typ :
		(
		HMIKEYCONSTATESTEP_DISABLED,
		HMIKEYCONSTATESTEP_STANDBY,
		HMIKEYCONSTATESTEP_HOME,
		HMIKEYCONSTATESTEP_CHANGEMODE,
		HMIKEYCONSTATESTEP_ACTIVE_JOG,
		HMIKEYCONSTATESTEP_ACTIVE_AUTO,
		HMIKEYCONSTATESTEP_ERROR
		);
	TcpFrameTest_typ : 	STRUCT
		X : LREAL;
		Y : LREAL;
		Z : LREAL;
		A : LREAL;
		B : LREAL;
		C : LREAL;
	END_STRUCT;
	SumInData_typ : 	STRUCT
		measure : UDINT;
		reserve_align0 : UDINT;
		P1 : TRF_FRAMEPOS_typ;
		dP : TRF_FRAMEPOS_typ;
		epsilon : LREAL;
		desired_phi : LREAL;
		desired_theta : LREAL;
		desired_psi : LREAL;
		angles_type : UDINT;
		reserve_align1 : UDINT;
	END_STRUCT;
	SumOutData_typ : 	STRUCT
		P2 : TRF_FRAMEPOS_typ;
	END_STRUCT;
	CreateInData_typ : 	STRUCT
		phi : LREAL;
		theta : LREAL;
		psi : LREAL;
		measure : UDINT;
		angles_type : UDINT;
		epsilon : LREAL;
	END_STRUCT;
	Angletypout_typ : 	STRUCT
		phi : LREAL;
		theta : LREAL;
		psi : LREAL;
	END_STRUCT;
	Angletyp2_typ : 	STRUCT
		phi : LREAL;
		theta : LREAL;
		psi : LREAL;
		measure : UDINT;
		angles_type1 : UDINT;
		angles_type2 : UDINT;
		reserve_align0 : UDINT;
		epsilon : LREAL;
		desired_phi : LREAL;
		desired_theta : LREAL;
		desired_psi : LREAL;
	END_STRUCT;
	HmiKeyCtrlHomeState_Type :
		(
		HOMESTATESTEP_COMMAND,
		HOMESTATESTEP_HOMING,
		HOMESTATESTEP_W_END
		);
	HmiKeyCtrlInternal_Type : 	STRUCT
		OldCommand : HmiKeyControlInputCommand_Type;
		HmiKeyControlState : HmiKeyControlStateSteps_Typ;
		HomeState : ARRAY[0..MAX_AX_MINUS_ONE]OF HmiKeyCtrlHomeState_Type;
		OldJogEnable : BOOL;
		OldRun : BOOL;
	END_STRUCT;
	CreateOutData_typ : 	STRUCT
		m11 : LREAL;
		m12 : LREAL;
		m13 : LREAL;
		m21 : LREAL;
		m22 : LREAL;
		m23 : LREAL;
		m31 : LREAL;
		m32 : LREAL;
		m33 : LREAL;
	END_STRUCT;
END_TYPE
```

### Package Logical/HmiHandling/HmiMain - Main Page

### HmiMainGlobal.typ - Global data types
```iecst
(********************************************************************
 * COPYRIGHT --
 ********************************************************************
 * Package: HmiMainNew
 * File: HmiMainGlobal.typ
 * Author: renj
 * Created: November 17, 2014
 ********************************************************************
 * Data types of package HmiMainNew
 ********************************************************************)

TYPE
	HmiMainCtrlComponentsType : 	STRUCT
		EditPrgRun : HmiEditType;
		TextFileName : HmiTextType;
		ButtonJumpToMain : HmiButtonType;
		HotSpotPrgRun : HmiSimpleType;
		ButtonSetPtr : HmiButtonType;
	END_STRUCT;
	HmiMainControlType : 	STRUCT
		Components : HmiMainCtrlComponentsType;
	END_STRUCT;
END_TYPE
```

### HmiMainGlobal.var - Global variables
```iecst
(********************************************************************
 * COPYRIGHT --
 ********************************************************************
 * Package: HmiMainNew
 * File: HmiMainGlobal.var
 * Author: renj
 * Created: November 17, 2014
 ********************************************************************
 * Variables of package HmiMainNew
 ********************************************************************)
VAR
	HmiMainCtrl : HmiMainControlType := (0);
END_VAR
```

### HmiFileGlobal.var - Global variables
```iecst
(********************************************************************
 * COPYRIGHT --
 ********************************************************************
 * Package: HmiFileCtrl
 * File: HmiFileCtrlGlobal.var
 * Author: renj
 * Created: October 29, 2014
 ********************************************************************
 * Variables of package HmiFileCtrl
 ********************************************************************)
VAR
	HmiFileCtrl : HmiFileCtrl_Type := (0);
END_VAR
```

### Program Logical/HmiHandling/HmiMain/HmiMain (ANSIC) - Main Page

#### HmiMain.cpp - Implementation code
```cpp
/********************************************************************
 * COPYRIGHT --
 ********************************************************************
 * Program: HmiMain
 * File: HmiMain.cpp
 * Author: renj
 * Created: November 17, 2014
 ********************************************************************
 * Implementation of program HmiMain
 ********************************************************************/

#include <bur/plctypes.h>
#include <string>
#include <fileio.h>
#include "CusLib.hpp"

#ifdef _DEFAULT_INCLUDES
#include <AsDefault.h>
#endif

using namespace std;

unsigned long bur_heap_size = 0xFFFFF;

string ConvBuf; // the Buffer for the Programs to be shown(including the Line No)
bool ClearDone;

void _INIT HmiMainInit(void)
{

}

void _CYCLIC HmiMainCyclic(void)
{
	/**                          Initialization                              **/
	if (HmiGlobal.PageControl.ActPage == PAGE_MAIN)
	{
		if ((HmiGlobal.Address.CncAddress != 0) && (HmiGlobal.Address.SystemAddress != 0))
		{
			pCnc = (Cnc_Type *)(HmiGlobal.Address.CncAddress);
			pSystem = (System_Type *)(HmiGlobal.Address.SystemAddress);

		} else
		{
			Internal.MainEditCtrlState = HMIMAIN_WAIT;
			return;
		}

		// Highlight line calc
		UINT ActCNCLine;
		if (atoi(pCnc->Output.Monitor.NcBlock.TextActual) > 0)
			ActCNCLine = (UINT)(atoi(pCnc->Output.Monitor.NcBlock.TextActual));

		size_t LineNo, Pos;

		string FileName;

		switch (Internal.MainEditCtrlState)
		{
			case HMIMAIN_WAIT:
				// Read the Program into Buffer
				if (strcmp(HmiRetain.HmiProgram.Name, "") != 0 && strcmp(HmiRetain.HmiProgram.Device, "") != 0)
				{
					memset(HmiMainCtrl.Components.EditPrgRun.StringBuffer, 0, sizeof(HmiMainCtrl.Components.EditPrgRun.StringBuffer));
					strcpy(HmiFileCtrl.Input.Parameter.FileDevice, HmiRetain.HmiProgram.Device);
					FileName.assign(HmiRetain.HmiProgram.Name);
					strcpy(HmiFileCtrl.Input.Parameter.FileName, FileName.append(".st").c_str());

					HmiFileCtrl.Input.Parameter.StringBufferAdr = (UDINT)Internal.StringBuffer;
					HmiFileCtrl.Input.Parameter.StringBufferSize = sizeof(Internal.StringBuffer);

					memset(Internal.StringBuffer, 0, sizeof(Internal.StringBuffer));
					HmiFileCtrl.Input.Command.Read = 1;

					HmiMainCtrl.Components.TextFileName.TextIndex = 1;

					Internal.MainEditCtrlState = HMIMAIN_READWAIT;

				} else // No Program Available and the Text is gonna be shown. Do ONLY ONCE!!! ClearDone is reset when leaving the Main Page
				{
					if (!ClearDone)
					{
						memset(HmiMainCtrl.Components.EditPrgRun.StringBuffer, 0, sizeof(HmiMainCtrl.Components.EditPrgRun.StringBuffer));
						strcpy(HmiMainCtrl.Components.EditPrgRun.StringBuffer, "No Program Available");
						HmiMainCtrl.Components.TextFileName.TextIndex = 0;
						ClearDone = 1;
					}
				}

				break;

			case HMIMAIN_READWAIT:
				// File Read is done by separate task HmiFile
				if (HmiFileCtrl.Input.Command.Read == 0)
				{
					if (HmiFileCtrl.Output.Status.ReadOK)
					{
						ConvBuf.assign(Internal.StringBuffer);
						Internal.MainEditCtrlState = HMIMAIN_READPROCESS;

					} else
						Internal.MainEditCtrlState = HMIMAIN_ERROR;
				}
				break;

			case HMIMAIN_READPROCESS: // After Reading the File, add the Line No.

				ConvBuf.insert(0, StringHelper::GetLineNoStr(1));

				Pos = 0;
				LineNo = 2;

				while(true)
				{
					// Find "\r\n" and add Line No
					Pos = ConvBuf.find("\r\n", Pos);

					if (Pos == string::npos)
					{
						break;

					} else
					{
						Pos = Pos + 2;
						ConvBuf.insert(Pos, StringHelper::GetLineNoStr(LineNo)); // Generate teh Line No in this style "0008"
						LineNo++;
					}
				}
				// Set the Value of StringBuffer
				memcpy(HmiMainCtrl.Components.EditPrgRun.StringBuffer, ConvBuf.data(), ConvBuf.size());

				Internal.MainEditCtrlState = HMIMAIN_LOADED;

				break;

			case HMIMAIN_LOADED:
				// To Make sure the cursor is always set on the first col
				if (HmiMainCtrl.Components.EditPrgRun.CursorCol != 1 && HmiMainCtrl.Components.EditPrgRun.CommandStatus == 0)
				{
					stringstream ss;
					ss << "goto col=1 line=" << HmiMainCtrl.Components.EditPrgRun.CursorLine;
					strcpy(HmiMainCtrl.Components.EditPrgRun.CommandRequest, ss.str().c_str());

					HmiMainCtrl.Components.EditPrgRun.CommandStatus = 1;

				}

				if (pCnc->Output.State.Moving == 1) // If Program is running, the Highlight cannot be set
				{
					if (ActCNCLine != 0
						&& HmiMainCtrl.Components.EditPrgRun.CursorLine != ActCNCLine ) // Always Point to the Actual CNC Line
					{
						stringstream ss;
						ss << "highlight line=" << ActCNCLine;
						strcpy(HmiMainCtrl.Components.EditPrgRun.CommandRequest, ss.str().c_str());

						HmiMainCtrl.Components.EditPrgRun.CommandStatus = 1;

						Internal.MainEditCtrlState = HMIMAIN_HIGHLIGHT_WAIT;
					}

					HmiMainCtrl.Components.HotSpotPrgRun.StatusDatapoint = 0;

				} else
				{
					// Make the Hotspot Disappear to allow the User to change the Highlight line
					HmiMainCtrl.Components.HotSpotPrgRun.StatusDatapoint = 1;

					// Make sure the Edit Components in Edit Mode so the User can change the Highlight Line
					if ((HmiMainCtrl.Components.EditPrgRun.StatusDatapoint & (16384)) == 16384 && // 16384 means focused
						(HmiMainCtrl.Components.EditPrgRun.StatusDatapoint & (32768)) == 0 &&  // 32768 means in Edit Mode
						HmiMainCtrl.Components.EditPrgRun.CommandStatus == 0) // When its not busy
					{
						stringstream ss; // Highlight the LINE "PROGRAM _MAIN " at very beginning
						ss << "highlight line=" << StringHelper::StringTo<int>(ConvBuf.substr(ConvBuf.find("PROGRAM _MAIN") - 5, 4));

						strcpy(HmiMainCtrl.Components.EditPrgRun.CommandRequest, ss.str().c_str());
						HmiMainCtrl.Components.EditPrgRun.CommandStatus = 1;

					}
					// When Jump to Main is pressed, highlight the Line "PROGRAM _MAIN"
					if (HmiMainCtrl.Components.ButtonJumpToMain.Value > HmiMainCtrl.Components.ButtonJumpToMain.OldValue)
					{
						stringstream ss;
						ss << "highlight line=" << StringHelper::StringTo<int>(ConvBuf.substr(ConvBuf.find("PROGRAM _MAIN") - 5, 4));

						strcpy(HmiMainCtrl.Components.EditPrgRun.CommandRequest, ss.str().c_str());

						HmiMainCtrl.Components.EditPrgRun.CommandStatus = 1;

						Internal.MainEditCtrlState = HMIMAIN_HIGHLIGHT_WAIT;

					}

					// WHEN current Cursor is between "PROGRAM _MAIN" and "END_PROGRAM", the Ptr can be set in this case
					if (HmiMainCtrl.Components.EditPrgRun.CursorLine > StringHelper::StringTo<int>(ConvBuf.substr(ConvBuf.find("PROGRAM _MAIN") - 5, 4)) &&
						HmiMainCtrl.Components.EditPrgRun.CursorLine < StringHelper::StringTo<int>(ConvBuf.substr(ConvBuf.find("END_PROGRAM") - 5, 4)))
					{	// Set the Program Ptr
						if (HmiMainCtrl.Components.ButtonSetPtr.Value > HmiMainCtrl.Components.ButtonSetPtr.OldValue)
						{
							HmiRetain.HmiProgram.Ptr = HmiMainCtrl.Components.EditPrgRun.CursorLine;
						}
					}

				}

				break;

			case HMIMAIN_HIGHLIGHT_WAIT: // Acutally the State is not Necessary but kept anyway

				if (HmiMainCtrl.Components.EditPrgRun.CommandStatus == 0)
				{
					Internal.MainEditCtrlState = HMIMAIN_LOADED;
				} else if (HmiMainCtrl.Components.EditPrgRun.CommandStatus == 65533 || HmiMainCtrl.Components.EditPrgRun.CommandStatus == 65534)
				{
					Internal.MainEditCtrlState = HMIMAIN_ERROR;
				}
				break;

			case HMIMAIN_ERROR:
				break;

		}

	} else
	{
		Internal.MainEditCtrlState = HMIMAIN_WAIT;
		ClearDone = 0; // Everytime leave the Page the ClearDone is reset
	}

	// Button Edge Detection
	HmiMainCtrl.Components.ButtonJumpToMain.OldValue = HmiMainCtrl.Components.ButtonJumpToMain.Value;
	HmiMainCtrl.Components.ButtonSetPtr.OldValue = HmiMainCtrl.Components.ButtonSetPtr.Value;

}
```

#### HmiMainLocal.typ - Local data types
```iecst
(********************************************************************
 * COPYRIGHT --
 ********************************************************************
 * Program: HmiMain
 * File: HmiMainLocal.typ
 * Author: renj
 * Created: November 17, 2014
 ********************************************************************
 * Local data types of program HmiMain
 ********************************************************************)

TYPE
	HmiMainCtrlInternal_Type : 	STRUCT
		MainEditCtrlState : HmiMainCtrlState_Type;
		StringBuffer : STRING[10000];
	END_STRUCT;
	HmiMainCtrlState_Type :
		(
		HMIMAIN_WAIT,
		HMIMAIN_READWAIT,
		HMIMAIN_READPROCESS,
		HMIMAIN_LOADED,
		HMIMAIN_HIGHLIGHT_WAIT,
		HMIMAIN_ERROR
		);
END_TYPE
```

#### HmiMainLocal.var - Local variables
```iecst
(********************************************************************
 * COPYRIGHT --
 ********************************************************************
 * Program: HmiMain
 * File: HmiMainLocal.var
 * Author: renj
 * Created: November 17, 2014
 ********************************************************************
 * Local variables of program HmiMain
 ********************************************************************)
VAR
	pSystem : REFERENCE TO System_Type;
	pCnc : REFERENCE TO Cnc_Type;
	Internal : HmiMainCtrlInternal_Type;
END_VAR
```

### Program Logical/HmiHandling/HmiMain/HmiFile (IEC) - Read/Write File Task

#### HmiFileCtrl.st - Implementation code
```iecst
(********************************************************************
 * COPYRIGHT --
 ********************************************************************
 * Program: HmiFile
 * File: HmiFileCtrl.st
 * Author: renj
 * Created: October 29, 2014
 ********************************************************************
 * Implementation of program HmiFile
 ********************************************************************)

PROGRAM _INIT

END_PROGRAM

PROGRAM _CYCLIC

	CASE Internal.State OF

		HMIFILE_IDLE:

			IF HmiFileCtrl.Input.Command.Read THEN

				Internal.State := HMIFILE_OPEN;
				HmiFileCtrl.Output.Status.ReadOK := FALSE;

			END_IF

			IF HmiFileCtrl.Input.Command.Write THEN

				Internal.State := HMIFILE_DELETE;

				HmiFileCtrl.Output.Status.WriteOK := FALSE;

			END_IF

		HMIFILE_OPEN:

			FileOpen_0.enable	:= TRUE;
			FileOpen_0.pDevice 	:= ADR(HmiFileCtrl.Input.Parameter.FileDevice);
			FileOpen_0.pFile 	:= ADR(HmiFileCtrl.Input.Parameter.FileName);
			FileOpen_0.mode 	:= fiREAD_WRITE;
			(* FB Call *)
			FileOpen_0();

			(* Get FBK output information *)
			Internal.FileIdent := FileOpen_0.ident;
			wStatus := FileOpen_0.status;

			IF (wStatus = 0) THEN

				Internal.State := HMIFILE_READ;

			ELSIF (wStatus <> 65535) THEN
				(* Verify status (20708 -> File doesn't exist) *)
				IF (wStatus = 20708) THEN

				END_IF

				IF (wStatus = 20799) THEN
					wError := FileIoGetSysError();
				END_IF

				IF HmiFileCtrl.Input.Command.Read THEN

					HmiFileCtrl.Input.Command.Read := FALSE;

				ELSIF HmiFileCtrl.Input.Command.Write THEN

					HmiFileCtrl.Input.Command.Write := FALSE;

				END_IF

				Internal.State := HMIFILE_ERROR;

			END_IF

		HMIFILE_READ:

			(**** Read data from file ****)
			(* Initialize file read structure *)
			FileReadEx_0.enable		:= TRUE;
			FileReadEx_0.ident     	:= Internal.FileIdent;
			FileReadEx_0.pDest     	:= HmiFileCtrl.Input.Parameter.StringBufferAdr;
			FileReadEx_0.len	   	:= HmiFileCtrl.Input.Parameter.StringBufferSize;

			(* Call FBK *)
			FileReadEx_0();
			(* Get status *)
			wStatus := FileReadEx_0.status;
			(* Verify status *)
			IF wStatus = 0 THEN

				Internal.FileByte := FileReadEx_0.bytesread;

				Internal.State := HMIFILE_CLOSE;

			ELSIF (wStatus <> 65535) THEN

				IF (wStatus = 20799) THEN
					wError := FileIoGetSysError();
				END_IF

				IF HmiFileCtrl.Input.Command.Read THEN

					HmiFileCtrl.Input.Command.Read := FALSE;

				ELSIF HmiFileCtrl.Input.Command.Write THEN

					HmiFileCtrl.Input.Command.Write := FALSE;

				END_IF

				Internal.State := HMIFILE_ERROR;

			END_IF

		HMIFILE_DELETE:
			(* Initialize file delete structure *)
			FileDelete_0.enable  := 1;
			FileDelete_0.pDevice := ADR(HmiFileCtrl.Input.Parameter.FileDevice);
			FileDelete_0.pName   :=ADR(HmiFileCtrl.Input.Parameter.FileName);
			(* Call FBK *)
			FileDelete_0();
			(* Get status *)
			wStatus := FileDelete_0.status;

			(* Verify status *)
			IF wStatus = 0 THEN
				Internal.State := HMIFILE_CREATE;
			ELSIF (wStatus <> 65535) THEN

				IF (wStatus = 20799) THEN
					wError := FileIoGetSysError();
				END_IF

				IF HmiFileCtrl.Input.Command.Write THEN

					HmiFileCtrl.Input.Command.Write := FALSE;

				END_IF

				Internal.State := HMIFILE_ERROR;

			END_IF

		HMIFILE_CREATE:
			(* Initialize file create structure *)
			FileCreate_0.enable  := 1;
			FileCreate_0.pDevice := ADR(HmiFileCtrl.Input.Parameter.FileDevice);
			FileCreate_0.pFile   := ADR(HmiFileCtrl.Input.Parameter.FileName);
			(* Call FBK *)
			FileCreate_0();
			(* Get FBK output information *)
			Internal.FileIdent := FileCreate_0.ident;
			wStatus := FileCreate_0.status;
			(* Verify status *)
			IF wStatus = 0 THEN
				Internal.State := HMIFILE_WRITE;
			ELSIF (wStatus <> 65535) THEN

				IF (wStatus = 20799) THEN
					wError := FileIoGetSysError();
				END_IF

				IF HmiFileCtrl.Input.Command.Write THEN

					HmiFileCtrl.Input.Command.Write := FALSE;

				END_IF

				Internal.State := HMIFILE_ERROR;

			END_IF

		HMIFILE_WRITE:
			(**** WRITE File ****)
			(* Initialize file close structure *)
			FileWriteEx_0.enable	:= TRUE;
			FileWriteEx_0.ident		:= Internal.FileIdent;

			FileWriteEx_0.len		:= HmiFileCtrl.Input.Parameter.StringBufferSize;
			FileWriteEx_0.pSrc		:= HmiFileCtrl.Input.Parameter.StringBufferAdr;;

			(* Call FBK *)
			FileWriteEx_0();

			(* Get status *)
			wStatus := FileWriteEx_0.status;

			(* Verify status *)
			IF wStatus = 0 THEN
				Internal.State := HMIFILE_CLOSE;
			ELSIF (wStatus <> 65535) THEN

				IF (wStatus = 20799) THEN
					wError := FileIoGetSysError();
				END_IF

				IF HmiFileCtrl.Input.Command.Read THEN

					HmiFileCtrl.Input.Command.Read := FALSE;

				ELSIF HmiFileCtrl.Input.Command.Write THEN

					HmiFileCtrl.Input.Command.Write := FALSE;

				END_IF

				Internal.State := HMIFILE_ERROR;

			END_IF

		HMIFILE_CLOSE:
			(**** Close file ****)
			(* Initialize file close structure *)
			FileClose_0.enable	:= TRUE;
			FileClose_0.ident	:= Internal.FileIdent;

			(* Call FBK *)
			FileClose_0();

			(* Get status *)
			wStatus := FileClose_0.status;

			IF wStatus = 0 THEN

				IF HmiFileCtrl.Input.Command.Read THEN

					HmiFileCtrl.Output.Status.ReadOK := TRUE;

					HmiFileCtrl.Input.Command.Read := FALSE;

				ELSIF HmiFileCtrl.Input.Command.Write THEN

					HmiFileCtrl.Output.Status.WriteOK := TRUE;

					HmiFileCtrl.Input.Command.Write := FALSE;

				END_IF

				Internal.State := HMIFILE_IDLE;

			ELSIF (wStatus <> 65535) THEN

				IF (wStatus = 20799) THEN
					wError := FileIoGetSysError();
				END_IF

				IF HmiFileCtrl.Input.Command.Read THEN

					HmiFileCtrl.Input.Command.Read := FALSE;

				ELSIF HmiFileCtrl.Input.Command.Write THEN

					HmiFileCtrl.Input.Command.Write := FALSE;

				END_IF

				Internal.State := HMIFILE_ERROR;

			END_IF

		HMIFILE_ERROR:

			IF HmiFileCtrl.Input.Command.AckError THEN

				HmiFileCtrl.Input.Command.AckError := 0;
				Internal.State := HMIFILE_IDLE;

			END_IF

	END_CASE

END_PROGRAM
```

#### HmiFileLocal.typ - Local data types
```iecst
(********************************************************************
 * COPYRIGHT --
 ********************************************************************
 * Program: HmiFile
 * File: HmiFileLocal.typ
 * Author: renj
 * Created: October 29, 2014
 ********************************************************************
 * Local data types of program HmiFile
 ********************************************************************)

TYPE
	HmiFileCtrlInternalState_Type :
		(
		HMIFILE_IDLE,
		HMIFILE_OPEN,
		HMIFILE_READ,
		HMIFILE_CLOSE,
		HMIFILE_CREATE,
		HMIFILE_DELETE,
		HMIFILE_WRITE,
		HMIFILE_ERROR
		);
	HmiFileCtrlInternal_Type : 	STRUCT
		State : HmiFileCtrlInternalState_Type;
		FileIdent : UDINT;
		FileByte : UDINT;
	END_STRUCT;
END_TYPE
```

### Package Logical/HmiHandling/HmiSetup - Setup Page

### HmiSetupGlobal.typ - Global data types
```iecst
(********************************************************************
 * COPYRIGHT --
 ********************************************************************
 * Package: HmiMain
 * File: HmiMainGlobal.typ
 * Author: renj
 * Created: September 25, 2014
 ********************************************************************
 * Data types of package HmiMain
 ********************************************************************)

TYPE
	HmiSetupControl_Type : 	STRUCT
		Components : HmiSetupComponentsType;
	END_STRUCT;
	HmiSetupCalibType : 	STRUCT
		LayerInfo : HmiSetupCalibInfoType;
		LayerDefault : HmiSetupCalibDefaultType;
	END_STRUCT;
	HmiSetupCalibInfoType : 	STRUCT
		Layer : HmiLayerType;
	END_STRUCT;
	HmiSetupCalibDefaultType : 	STRUCT
		Layer : HmiLayerType;
		ButtonAxisRefresh : ARRAY[0..5]OF HmiButtonType;
		ButtonAxisToggle : ARRAY[0..5]OF HmiButtonType;
		NumericEncoderValue : ARRAY[0..5]OF HmiNumericType;
		ButtonSave : HmiButtonType;
	END_STRUCT;
	HmiSetupMainDefaultType : 	STRUCT
		HotspotRestart : HmiHotSpotType;
		Layer : HmiLayerType;
	END_STRUCT;
	HmiSetupMainInfoType : 	STRUCT
		Layer : HmiLayerType;
		ButtonRestart : HmiButtonType;
	END_STRUCT;
	HmiSetupMainType : 	STRUCT
		LayerInfo : HmiSetupMainInfoType;
		LayerDefault : HmiSetupMainDefaultType;
	END_STRUCT;
	HmiSetupComponentsType : 	STRUCT
		PageCalib : HmiSetupCalibType;
		PageKine : HmiSetupKineType;
		PageMain : HmiSetupMainType;
	END_STRUCT;
	HmiSetupKineDefaultType : 	STRUCT
		ButtonSave : HmiButtonType;
		NumericC56Value : HmiNumericType;
		NumericC46Value : HmiNumericType;
		NumericC45Value : HmiNumericType;
		ButtonC56Enable : HmiButtonType;
		ButtonC46Enable : HmiButtonType;
		ButtonC45Enable : HmiButtonType;
		DropdownAxisSelect : HmiDropdownType;
	END_STRUCT;
	HmiSetupKineInfoType : 	STRUCT
		Layer : HmiLayerType;
	END_STRUCT;
	HmiSetupKineType : 	STRUCT
		LayerDefault : HmiSetupKineDefaultType;
		LayerInfo : HmiSetupKineInfoType;
	END_STRUCT;
END_TYPE
```

### HmiSetupGlobal.var - Global variables
```iecst
(********************************************************************
 * COPYRIGHT --
 ********************************************************************
 * Package: HmiMain
 * File: HmiMainGlobal.var
 * Author: renj
 * Created: September 25, 2014
 ********************************************************************
 * Variables of package HmiMain
 ********************************************************************)
VAR
	HmiSetupCtrl : HmiSetupControl_Type := (0);
END_VAR
```

### HmiSetupLocalGlobal.var - Global variables
```iecst
(********************************************************************
 * COPYRIGHT --
 ********************************************************************
 * Package: HmiEdit
 * File: HmiEditGlobal.var
 * Author: renj
 * Created: October 20, 2014
 ********************************************************************
 * Variables of package HmiEdit
 ********************************************************************)
VAR
	HmiFileTools : HmiFileCtrl_Type := (0);
END_VAR
```

### Program Logical/HmiHandling/HmiSetup/HmiSetup (ANSIC) - Setup Page

#### HmiSetupCtrl.cpp - Implementation code
```cpp
/********************************************************************
 * COPYRIGHT --
 ********************************************************************
 * Program: HmiSetup
 * File: HmiSetupCtrl.cpp
 * Author: renj
 * Created: January 21, 2015
 ********************************************************************
 * Implementation of program HmiSetup
 ********************************************************************/

#include <bur/plctypes.h>
#include <string.h>

#ifdef _DEFAULT_INCLUDES
	#include <AsDefault.h>
#endif

unsigned long bur_heap_size = 0xFFFFF;

void _INIT HmiSetupCtrlInit(void)
{
	HmiSetupCtrl.Components.PageCalib.LayerInfo.Layer.StatusDatapoint = 1;
	HmiSetupCtrl.Components.PageKine.LayerInfo.Layer.StatusDatapoint = 1;
	HmiSetupCtrl.Components.PageMain.LayerInfo.Layer.StatusDatapoint = 1;
}

int HomeStep;
int AxisIndex;
UINT OldPage;

void _CYCLIC HmiSetupCtrlCyclic(void)
{
	if (HmiGlobal.Address.AxesAddress != 0 && HmiGlobal.Address.RecipeAddress != 0 && HmiGlobal.Address.SystemAddress)
	{
		pSystem = (System_Type *) HmiGlobal.Address.SystemAddress;
		pAxes = (Axes_Type (*) [13])HmiGlobal.Address.AxesAddress;
		pRecipe = (RECIPE_typ *) HmiGlobal.Address.RecipeAddress;
	} else
		return;

	// Page Calibration
	if (HmiGlobal.PageControl.ActPage == PAGE_SETUPCALIB && HmiKeyControl.Output.Status.MoveStatus == LOCK)	// Move Single Axis without SW Limits only allowed in Setup Calib Page when axes is select
	{
		// Handle the Toggle of Exclusive Checkbox Group
		for (int i = 0; i < 6; ++i)
			{
			if (HmiSetupCtrl.Components.PageCalib.LayerDefault.ButtonAxisToggle[i].Value > HmiSetupCtrl.Components.PageCalib.LayerDefault.ButtonAxisToggle[i].OldValue)
			{
				for (int j = 0; j < 6; ++ j)
					if (j != i)
					HmiSetupCtrl.Components.PageCalib.LayerDefault.ButtonAxisToggle[j].Value = 0;

			}
		}
		// SW limit ignore control only when toggled, the Limit is ignored
		for (int i = 0; i < 6; ++i)
			{
			if (HmiSetupCtrl.Components.PageCalib.LayerDefault.ButtonAxisToggle[i].Value == 1)
			{
				if (!HmiKeyControl.Output.Status.SWLimitsIgnored[i])
				{
					(*pAxes)[i+6].Input.Parameter.WriteParID = ACP10PAR_SGEN_SW_END_IGNORE;
					strcpy((*pAxes)[i+6].Input.Parameter.WriteParIDText,  "1");
					(*pAxes)[i+6].Input.Command.WriteAxisPar = 1;
					HmiKeyControl.Output.Status.SWLimitsIgnored[i] = 1;
				}
			} else
			{
				if (HmiKeyControl.Output.Status.SWLimitsIgnored[i])
				{
					(*pAxes)[i+6].Input.Parameter.WriteParID = ACP10PAR_SGEN_SW_END_IGNORE;
					strcpy((*pAxes)[i+6].Input.Parameter.WriteParIDText,  "0");
					(*pAxes)[i+6].Input.Command.WriteAxisPar = 1;
					HmiKeyControl.Output.Status.SWLimitsIgnored[i] = 0;
				}
			}
		}

		// Encoder Value Update
		switch (HomeStep)
		{
			case 0: // Do the Homing with Homeposition 0 to get the REAL Homeposiiton
				for (int i = 0; i < 6; ++i)
					{
					if (HmiSetupCtrl.Components.PageCalib.LayerDefault.ButtonAxisToggle[i].Value == 1)
					{
						if (HmiSetupCtrl.Components.PageCalib.LayerDefault.ButtonAxisRefresh[i].Value > HmiSetupCtrl.Components.PageCalib.LayerDefault.ButtonAxisRefresh[i].Value
							&& !(*pAxes)[i+6].Output.State.Homing &&  !(*pAxes)[i+6].Output.Status.Busy)
						{
							(*pAxes)[i+6].Input.Parameter.HomePosition = 0;
							(*pAxes)[i+6].Input.Command.Home = 1;
							AxisIndex = i;
							HomeStep = 1;
						}
					}
				}
				break;

			case 1:
				if (!(*pAxes)[AxisIndex+6].Output.State.Homing && !(*pAxes)[AxisIndex+6].Output.Status.Busy)
					HmiSetupCtrl.Components.PageCalib.LayerDefault.NumericEncoderValue[AxisIndex].Value = (*pAxes)[AxisIndex+6].Output.Monitor.Position;

				HomeStep = 0;
				break;
		}

	} else
	{
		// If in other Page or In other Mode, SW Limits is not Ignored
		for (int i = 0; i < 6; ++i)
		{
			HmiSetupCtrl.Components.PageCalib.LayerDefault.ButtonAxisToggle[i].Value = 0;

			if (HmiKeyControl.Output.Status.SWLimitsIgnored[i])
			{
				(*pAxes)[i+6].Input.Parameter.WriteParID = ACP10PAR_SGEN_SW_END_IGNORE;
				strcpy((*pAxes)[i+6].Input.Parameter.WriteParIDText,  "0");
				(*pAxes)[i+6].Input.Command.WriteAxisPar = 1;
				HmiKeyControl.Output.Status.SWLimitsIgnored[i] = 0;
			}
		}

		HomeStep = 0;
	}

	// But its not mandatory to be in lock mode to "SAVE" the Homeposition
	if (HmiGlobal.PageControl.ActPage == PAGE_SETUPCALIB)
	{
		if (OldPage != PAGE_SETUPCALIB)
			for (int i = 0; i < 6; ++i)
			HmiSetupCtrl.Components.PageCalib.LayerDefault.NumericEncoderValue[i].Value = - pRecipe->Data.System.HomePosition[i];

		// Save the HomePosition
		if (HmiSetupCtrl.Components.PageCalib.LayerDefault.ButtonSave.Value > HmiSetupCtrl.Components.PageCalib.LayerDefault.ButtonSave.OldValue)
		{
			for (int i = 0; i < 6; ++i)
				pRecipe->Data.System.HomePosition[i] = -HmiSetupCtrl.Components.PageCalib.LayerDefault.NumericEncoderValue[i].Value;
			pRecipe->Cmd.SysDataWrite = 1;

			HmiRetain.HmiKeyControl.MechHomeOK = 1;

		}
	}

	// Page Kinematics
	if (HmiGlobal.PageControl.ActPage == PAGE_SETUPKINEMATICS)
	{
		// First Come to the Page Setup Kinematics
		if (OldPage != PAGE_SETUPKINEMATICS)
		{
			//Some Initialization and Loading of Values
			HmiSetupCtrl.Components.PageKine.LayerInfo.Layer.StatusDatapoint = 1;

			HmiSetupCtrl.Components.PageKine.LayerDefault.ButtonC45Enable.Value = HmiRetain.HmiRobot.Coupling[0].Enable;
			HmiSetupCtrl.Components.PageKine.LayerDefault.NumericC45Value.Value = HmiRetain.HmiRobot.Coupling[0].Coefficient;
			HmiSetupCtrl.Components.PageKine.LayerDefault.ButtonC56Enable.Value = HmiRetain.HmiRobot.Coupling[1].Enable;
			HmiSetupCtrl.Components.PageKine.LayerDefault.NumericC56Value.Value = HmiRetain.HmiRobot.Coupling[1].Coefficient;
			HmiSetupCtrl.Components.PageKine.LayerDefault.ButtonC46Enable.Value = HmiRetain.HmiRobot.Coupling[2].Enable;
			HmiSetupCtrl.Components.PageKine.LayerDefault.NumericC46Value.Value = HmiRetain.HmiRobot.Coupling[2].Coefficient;

			HmiSetupCtrl.Components.PageKine.LayerDefault.DropdownAxisSelect.SelectedIndex = 0;

			for (int i = 0; i < 6; ++i)
			{
				KineAxes[i].Mech.Direction = HmiRetain.HmiRobot.Mech[i].Direction;

				KineAxes[i].JointLimits.Max = HmiRetain.HmiRobot.JointLimits[i].Max;
				KineAxes[i].JointLimits.Min = HmiRetain.HmiRobot.JointLimits[i].Min;
				KineAxes[i].Mech.OffsetX = HmiRetain.HmiRobot.Mech[i].OffsetX;
				KineAxes[i].Mech.OffsetY = HmiRetain.HmiRobot.Mech[i].OffsetY;
				KineAxes[i].Mech.OffsetZ = HmiRetain.HmiRobot.Mech[i].OffsetZ;

			}
		}
		// Using Pointer to access the seleted Axis
		pKineAxis = &(KineAxes[HmiSetupCtrl.Components.PageKine.LayerDefault.DropdownAxisSelect.SelectedIndex]);

		// Save the Coupling and Geometry
		if (HmiSetupCtrl.Components.PageKine.LayerDefault.ButtonSave.Value > HmiSetupCtrl.Components.PageKine.LayerDefault.ButtonSave.OldValue)
		{
			HmiSetupCtrl.Components.PageKine.LayerInfo.Layer.StatusDatapoint = 0;

			HmiRetain.HmiRobot.Coupling[0].Enable = HmiSetupCtrl.Components.PageKine.LayerDefault.ButtonC45Enable.Value;
			HmiRetain.HmiRobot.Coupling[0].Coefficient = HmiSetupCtrl.Components.PageKine.LayerDefault.NumericC45Value.Value;
			HmiRetain.HmiRobot.Coupling[1].Enable = HmiSetupCtrl.Components.PageKine.LayerDefault.ButtonC56Enable.Value;
			HmiRetain.HmiRobot.Coupling[1].Coefficient = HmiSetupCtrl.Components.PageKine.LayerDefault.NumericC56Value.Value;
			HmiRetain.HmiRobot.Coupling[2].Enable = HmiSetupCtrl.Components.PageKine.LayerDefault.ButtonC46Enable.Value;
			HmiRetain.HmiRobot.Coupling[2].Coefficient = HmiSetupCtrl.Components.PageKine.LayerDefault.NumericC46Value.Value;

			for (int i = 0; i < 6; ++i)
				{
				HmiRetain.HmiRobot.Mech[i].Direction = KineAxes[i].Mech.Direction;

				HmiRetain.HmiRobot.JointLimits[i].Max = KineAxes[i].JointLimits.Max;
				HmiRetain.HmiRobot.JointLimits[i].Min = KineAxes[i].JointLimits.Min;
				HmiRetain.HmiRobot.Mech[i].OffsetX = KineAxes[i].Mech.OffsetX;
				HmiRetain.HmiRobot.Mech[i].OffsetY = KineAxes[i].Mech.OffsetY;
				HmiRetain.HmiRobot.Mech[i].OffsetZ = KineAxes[i].Mech.OffsetZ;

			}

		}

	} else
	{

	}

	// Page Setup Main
	if (HmiGlobal.PageControl.ActPage == PAGE_SETUP)
	{
		// Visual Control
		if (OldPage != PAGE_SETUP)
		{
			HmiSetupCtrl.Components.PageMain.LayerInfo.Layer.StatusDatapoint = 1;
		}

		if (HmiSetupCtrl.Components.PageMain.LayerDefault.HotspotRestart.Value > HmiSetupCtrl.Components.PageMain.LayerDefault.HotspotRestart.OldValue)
		{
			HmiSetupCtrl.Components.PageMain.LayerInfo.Layer.StatusDatapoint = 0;
		}

		// Restart Button
		if (HmiSetupCtrl.Components.PageMain.LayerInfo.ButtonRestart.Value > HmiSetupCtrl.Components.PageMain.LayerInfo.ButtonRestart.OldValue)
		{
			SYSreset(1, 1);
		}
	}

	// PosEdge Detecting using programming way
	for (int i = 0; i < 6; ++i)
	{
		HmiSetupCtrl.Components.PageCalib.LayerDefault.ButtonAxisRefresh[i].OldValue = HmiSetupCtrl.Components.PageCalib.LayerDefault.ButtonAxisRefresh[i].Value;
		HmiSetupCtrl.Components.PageCalib.LayerDefault.ButtonAxisToggle[i].OldValue = HmiSetupCtrl.Components.PageCalib.LayerDefault.ButtonAxisToggle[i].Value;
	}

	HmiSetupCtrl.Components.PageCalib.LayerDefault.ButtonSave.OldValue = HmiSetupCtrl.Components.PageCalib.LayerDefault.ButtonSave.Value;

	HmiSetupCtrl.Components.PageKine.LayerDefault.ButtonSave.OldValue = HmiSetupCtrl.Components.PageKine.LayerDefault.ButtonSave.Value;

	HmiSetupCtrl.Components.PageMain.LayerDefault.HotspotRestart.OldValue = HmiSetupCtrl.Components.PageMain.LayerDefault.HotspotRestart.Value;
	HmiSetupCtrl.Components.PageMain.LayerInfo.ButtonRestart.OldValue = HmiSetupCtrl.Components.PageMain.LayerInfo.ButtonRestart.Value;

	OldPage = HmiGlobal.PageControl.ActPage;

}
```

#### HmiSetupLocal.typ - Local data types
```iecst
(********************************************************************
 * COPYRIGHT --
 ********************************************************************
 * Program: HmiSetup
 * File: HmiSetupLocal.typ
 * Author: renj
 * Created: January 21, 2015
 ********************************************************************
 * Local data types of program HmiSetup
 ********************************************************************)

TYPE
	KineAxisType : 	STRUCT
		Mech : HmiMechType;
		JointLimits : HmiJointLimitType;
	END_STRUCT;
END_TYPE
```

#### HmiSetupLocal.var - Local variables
```iecst
(********************************************************************
 * COPYRIGHT --
 ********************************************************************
 * Program: HmiSetup
 * File: HmiSetupLocal.var
 * Author: renj
 * Created: January 21, 2015
 ********************************************************************
 * Local variables of program HmiSetup
 ********************************************************************)
VAR
	pSystem : REFERENCE TO System_Type;
	pRecipe : REFERENCE TO RECIPE_typ;
	pAxes : REFERENCE TO ARRAY[0..12] OF Axes_Type;
	pKineAxis : REFERENCE TO KineAxisType;
	KineAxes : ARRAY[0..5] OF KineAxisType := [6(0)];
	test : ARRAY[0..21] OF USINT := [0,2,3,19(0)];
	New_Variable : ARRAY[0..1] OF BOOL := [2(TRUE)];
END_VAR
```

### Package Logical/HmiHandling/HmiIO - IO Page(NOT USED)

### HmiIOGlobal.typ - Local data types
```iecst
(********************************************************************
 * COPYRIGHT -- Bernecker + Rainer
 ********************************************************************
 * Program: HmiDiagnostics
 * File: HmiDiagnostics.typ
 * Author: B&R, International Applications
 * Created: February 13, 2009
 ********************************************************************
 * Local data types of program HmiDiagnostics
 ********************************************************************)

TYPE
	HmiIOCtrl_Type : 	STRUCT
		Input : HmiIOCtrlInput_Type;
		Output : HmiIOCtrlOutput_Type;
	END_STRUCT;
	HmiIOCtrlInputCommand_Type : 	STRUCT
		InfoLineUp : BOOL;
		InfoLineDown : BOOL;
		Enter : BOOL;
		DiscardChange : BOOL;
		ForcingOn : BOOL;
		ForcingOff : BOOL;
		ForcingAllOff : BOOL;
		SetValue : BOOL;
		PageUp : BOOL;
		PageDown : BOOL;
	END_STRUCT;
	HmiIOCtrlInput_Type : 	STRUCT
		Command : HmiIOCtrlInputCommand_Type;
	END_STRUCT;
	HmiIOCtrlOutput_Type : 	STRUCT
		ModuleInfo : HmiIOCtrlOutputModuleDiag_Type;
		IOInfo : HmiIOCtrlOutputIODiag_Type;
		Status : HmiIOCtrlOutputStatus_Type;
	END_STRUCT;
	HmiIOCtrlOutputModuleDiag_Type : 	STRUCT
		ModuleName : ARRAY[0..MAX_LINES_MINUS_ONE]OF STRING[20]; (*module name*)
		ModulePath : ARRAY[0..MAX_LINES_MINUS_ONE]OF STRING[30]; (*module path*)
		ModuleState : ARRAY[0..MAX_LINES_MINUS_ONE]OF USINT; (*module state*)
		ErrorModuleName : ARRAY[0..MAX_LINES_MINUS_ONE]OF STRING[20]; (*error module name*)
		Color : ARRAY[0..MAX_LINES_MINUS_ONE]OF UINT; (*color of each row*)
		WrongModulStatus : ARRAY[0..MAX_LINES_MINUS_ONE]OF USINT; (*wrong module inserted status*)
	END_STRUCT;
	HmiIOCtrlOutputIODiag_Type : 	STRUCT
		ModuleName : STRING[20]; (*module name*)
		ModulePath : STRING[30]; (*module path*)
		ModuleStatus : USINT; (*module status*)
		PVName : ARRAY[0..MAX_IO_LINES_MINUS_ONE]OF STRING[64]; (*PV names*)
		LogicalName : ARRAY[0..MAX_IO_LINES_MINUS_ONE]OF STRING[32]; (*logical names*)
		DiagnosicsType : ARRAY[0..MAX_IO_LINES_MINUS_ONE]OF USINT; (*data type*)
		ActValue : ARRAY[0..MAX_IO_LINES_MINUS_ONE]OF DINT; (*actual value*)
		ForceValue : ARRAY[0..MAX_IO_LINES_MINUS_ONE]OF DINT; (*force value*)
		MinValue : ARRAY[0..MAX_IO_LINES_MINUS_ONE]OF DINT; (*minimum value*)
		MaxValue : ARRAY[0..MAX_IO_LINES_MINUS_ONE]OF DINT; (*maximum value*)
		Color : ARRAY[0..MAX_IO_LINES_MINUS_ONE]OF UINT; (*color of each row*)
		NumericColor : ARRAY[0..MAX_IO_LINES_MINUS_ONE]OF UINT; (*color for numeric fields*)
		EnableForcing : ARRAY[0..MAX_IO_LINES_MINUS_ONE]OF BOOL; (*enable forcing*)
		InivisibleLines : ARRAY[0..MAX_IO_LINES_MINUS_ONE]OF USINT; (*hide rows datapoint*)
		CompletionCmdForcing : BOOL; (*completion datapoint for forcing button*)
		SelectedIO : HmiIOCtrlSelected_Type;
	END_STRUCT;
	HmiIOCtrlSelected_Type : 	STRUCT
		LogicalName : STRING[40];
		PVName : STRING[64];
		ForceValue : DINT;
		MinValue : DINT;
		MaxValue : DINT;
		Status : UINT;
	END_STRUCT;
	HmiIOCtrlOutputStatus_Type : 	STRUCT
		IOInformationStatus : USINT;
		SimulationActive : BOOL;
		DiagnosticsInitDone : BOOL;
		PageFocusColor : UINT; (*page focus color datapoint*)
		Address : UDINT;
		IOForced : USINT;
		ModuleInfoLayerStatus : USINT; (*runitme datapoint of module information layer*)
		IOInfoLayerStatus : USINT; (*runtime datapoint of I/O info layer*)
		StatusLayerMessage : USINT; (*runtime datapoint of warning message layer*)
	END_STRUCT;
	ModuleInformation_Type : 	STRUCT
		ModulePath : STRING[30]; (*module path*)
		ModuleName : STRING[20]; (*module name*)
		ModuleState : USINT; (*module state*)
		ModuleColor : USINT; (*module color*)
		ErrorModuleName : STRING[20]; (*name of module with error*)
	END_STRUCT;
	HW_DI_typ : 	STRUCT
		I1 : BOOL;
		I2 : BOOL;
		I3 : BOOL;
		I4 : BOOL;
		I5 : BOOL;
		I6 : BOOL;
		I7 : BOOL;
		I8 : BOOL;
		I9 : BOOL;
		I10 : BOOL;
		I11 : BOOL;
		I12 : BOOL;
		I13 : BOOL;
		I14 : BOOL;
		I15 : BOOL;
		I16 : BOOL;
	END_STRUCT;
	HW_DO_typ : 	STRUCT
		O1 : BOOL;
		O2 : BOOL;
		O3 : BOOL;
		O4 : BOOL;
		O5 : BOOL;
		O6 : BOOL;
		O7 : BOOL;
		O8 : BOOL;
		O9 : BOOL;
		O10 : BOOL;
		O11 : BOOL;
		O12 : BOOL;
		O13 : BOOL;
		O14 : BOOL;
		O15 : BOOL;
		O16 : BOOL;
	END_STRUCT;
END_TYPE
```

### HmiIOGlobal.var
```iecst
(********************************************************************
 * COPYRIGHT -- Bernecker + Rainer
 ********************************************************************
 * Program: HmiDiagnostics
 * File: HmiDiagnostics.var
 * Author: B&R, International Applications
 * Created: February 13, 2009
 ********************************************************************
 * Local variables of program HmiDiagnostics
 ********************************************************************)
VAR CONSTANT
	MAX_LINES : USINT := 21;
	MAX_LINES_MINUS_ONE : USINT := MAX_LINES-1;
	MAX_IO_LINES_MINUS_ONE : USINT := MAX_IO_LINES-1;
	MAX_IO_LINES : USINT := 15;
END_VAR
VAR
	HmiIOCtrl : HmiIOCtrl_Type;
	DI1 : HW_DI_typ := (0);
	DI2 : HW_DI_typ := (0);
	DI3 : HW_DI_typ := (0);
	DI4 : HW_DI_typ := (0);
	DI5 : HW_DI_typ := (0);
	DO1 : HW_DO_typ := (0);
	DO2 : HW_DO_typ := (0);
	DO3 : HW_DO_typ := (0);
	DO4 : HW_DO_typ := (0);
	DO5 : HW_DO_typ := (0);
END_VAR
```

### Package Logical/HmiHandling/HmiIO/Doc - Documentation

- TaskInteractionDiagnostics.vsd (binary file, 136704 bytes)
### Library Logical/HmiHandling/HmiIO/ModDiag (ANSIC, version 2.02.0)
Depends on: AsIO, AsIODiag, AsIOMMan, Sys_lib, Standard, DataObj

#### ModDiag.fun
```iecst
FUNCTION_BLOCK ModuleDiagnose
	VAR_INPUT
		AdrModuleInformationBuffer	:UDINT;
		Option	:USINT;
		AdrAlarmInformation	:UDINT;
	END_VAR
	VAR_OUTPUT
		status	:UINT;
	END_VAR
	VAR
		ActualModuleInformation	:SingleModuleInformationData_typ;
		PathBuffer	:ARRAY[0..99] OF STRING[30];
		Step	:USINT;
		LastStep	:USINT;
		NumberOfTotalModules	:USINT;
		ModuleIndex	:USINT;
		ModuleNumber	:USINT;
		ModulesLastCheck	:USINT;
		NumberNotCheckedModules	:USINT;
		ModuleDifference	:USINT;
		ResetModuleAlarms	:USINT;
		WaitTimer	:TON;
	END_VAR
END_FUNCTION_BLOCK
FUNCTION IOStatus : UINT
	VAR_INPUT
		pIOList	:UDINT;
		pStatusBuffer	:UDINT;
		Elements	:UINT;
		pEnableForce	:UDINT;
		pForceValue	:UDINT;
	END_VAR
END_FUNCTION
FUNCTION IOList : UINT
	VAR_INPUT
		pIOInformation	:UDINT;
	END_VAR
END_FUNCTION
```

#### ModDiag.typ
```iecst
TYPE
	IODPList_typ : STRUCT
		StartAdrBuffer	: UDINT ;
		NumberDigitalInput	: UINT ;
		NumberDigitalOutput	: UINT ;
		NumberAnalogInput	: UINT ;
		NumberAnalogOutput	: UINT ;
		TotalIONumber	: UINT ;
	END_STRUCT;
	SingleIOEntry_typ : STRUCT
		ModuleName	: STRING[20] ;
		Device	: STRING[60] ;
		ID	: STRING[60] ;
		LogicalName	: STRING[40] ;
		Type	: USINT ;
		PVName	: STRING[512] ;
	END_STRUCT;
	SingleIOStatus_typ : STRUCT
		ForceActive	: BOOL ;
		ActForceValue	: DINT ;
		ActValue	: DINT ;
		DataType	: USINT ;
	END_STRUCT;
	ModuleAlarmInformation_typ : STRUCT
		ErrorModulePath	: STRING[30] ;
		ErrorModuleName	: STRING[20] ;
		AlarmBitField	: ARRAY[0..299] OF BOOL ;
		ACKBitField	: ARRAY[0..299] OF BOOL ;
	END_STRUCT;
	SingleModuleInformationData_typ : STRUCT
		ModulePath	: STRING[30] ;
		ModuleName	: STRING[20] ;
		ModuleState	: USINT ;
		ModuleColor	: USINT ;
		ErrorModuleName	: STRING[20] ;
	END_STRUCT;
	ModuleInformationBuffer_typ : STRUCT
		ModuleInformation	: ARRAY[0..99] OF SingleModuleInformationData_typ ;
	END_STRUCT;
END_TYPE
```

#### ModDiag.var
```iecst
VAR CONSTANT
	MAX_MODULE_NUMBER	: UINT	:= 100;
END_VAR
```

#### internal_h.h
```c
typedef struct	SingleModuleInfo
{
	STRING	ModuleName[20];
	STRING	ModulePath[40];
}SingleModuleInfo_typ;

typedef struct	ModuleInfo
{
	USINT	Step;
	UDINT	HWIdent;
	UDINT	ModuleIndex;
	UDINT	TotalModules;
	UDINT	StartAdrBuffer;
	UDINT	IgnoredModules;
}ModuleInfo_typ;

typedef struct	IOStringInfo
{
	STRING	ModuleName[20];
	STRING	Device[60];
	STRING	ID[60];
	STRING	LogicalName[40];
	USINT	Type;
	STRING	PVName[512];
}IOStringInfo_typ;

typedef struct IOCounter
{
	UINT	NumberDigitalInputs;
	UINT	NumberDigitalOutputs;
	UINT	NumberAnalogInputs;
	UINT	NumberAnalogOutputs;
}IOCounter_typ;
```
